(* CoDeSys 2.3 library: oscat270.lib *)
(* Libraries: Standard.lib 22.11.04 11:21:12, SYSLIBCALLBACK.LIB 20.4.05 10:04:48 *)

(* Global variable list: Constants *)
VAR_GLOBAL CONSTANT
	(* setup Parameters *)
	STEP7 : BOOL := FALSE;

	(* Mathematische Konstanten *)
	PI1 : REAL := 3.14159265358979323846264338327950288;	(* Kreiszahl PI *)
	PI2 : REAL := 6.283185307179586476;					(* PI * 2 *)
	E : REAL := 2.71828182845904523536028747135266249;	(* Eulersche Konstante *)

	(* Physikalische Konstanten *)
	C0 : REAL := 299792458 ;							(* Lichtgeschwindigkeit in m/s *)
	EL : REAL := 1.60217653E-19;						(* elementarladung in Colomb = A * s *)
	GN : REAL := 9.80665; 								(* Erdbeschleunigung in m / s² *)
	TK : REAL := -273.15;									(* absoluter Nullpunkt in °C *)
	RU : REAL := 8.314472; 								(*Universelle Gaskonstante in J / (mol · K) *)
	PN : REAL := 101325;									(* NormalDruck in Pa *)

END_VAR

VAR_GLOBAL
END_VAR

(* revisionhistory
hm 3.3.2007
	extended accuracy of pi2
	renamed T0 to Tk for better compatibility with other libraries
	renamed C t0 c0 for better compatibility

hm	2.5.2007
	added RU universal gas constant

hm	1. oct 2007
	added setup parameter STEP7

hm 31. oct 2007
	added PN
*)

(* Data type *)
TYPE esr_data :
STRUCT
	typ : BYTE;
	adress : STRING(10);
	DS : DT;
	TS : TIME;
	data : ARRAY[0..7] OF BYTE;
END_STRUCT
END_TYPE

(* Data type *)
TYPE vector_3 :
STRUCT
	X : REAL;
	Y : REAL;
	Z : REAL;
END_STRUCT
END_TYPE

(* POU _array_init, ST *)
FUNCTION _array_init : BOOL
VAR_INPUT
	pt : POINTER TO ARRAY[0..32000] OF REAL;
	size : INT;
	init : REAL;
END_VAR
VAR
	i: INT;
	stop: INT;
END_VAR


(*
version 1.2	14 nov 2007
programmer 	hugo
tested by		tobias

this function will initialize a given array with a value init.
the function needs to be called:	_array_init(adr("array"),sizeof("array"));
this function will manipulate a given array.
the function manipulates the original array, it rerturnes true when finished.
because this function works with pointers its very time efficient and it needs no extra memory.

*)
stop := SHR(size,2)-1;
FOR i := 0 TO stop DO
	pt^[i] := init;
END_FOR;

_array_init := TRUE;

(* revision History

hm 6.1.2007		rev 1.1
	change type of function to bool
	added  array_init := true to set output true.

hm	14.11.2007	rev 1.2
	changed stop calculation to be more efficient
*)
END_FUNCTION

(* POU _array_median, ST *)
FUNCTION _array_median : REAL
VAR_INPUT
	pt : POINTER TO ARRAY[0..32000] OF REAL;
	size : INT;
END_VAR
VAR
	i: INT;
	stop: INT;
END_VAR

(*
version 1.4	14 nov 2007
programmer 	hugo
tested by		tobias

this function will calculate the median of a given array.
in order to do so the ariginal array is sorted and stays sorted after the function finishes
the function needs to be called:	_array_median(adr("array"),sizeof("array"));
this function will manipulate a given array.
the function will return the median of the original array.
for example [12,0,4,7,1] the median is 4 and the array after the function is called is [0,1,4,7,12]
because this function works with pointers its very time efficient and it needs no extra memory.

*)
_array_sort(pt,size);
stop := SHR(size,2)-1;
IF even(stop) THEN
	_array_median := pt^[stop/2];
ELSE
	i := SHR(stop,1);
	_array_median := (pt^[i] + pt^[i+1]) / 2;
END_IF;

(* old code
stop := (size - SIZEOF(pt)) / SIZEOF(pt);
FOR i := 0 TO stop - 1 DO
	FOR m := i + 1 TO stop DO
		IF pt^[i] > pt^[m] THEN
			temp := pt^[i];
			pt^[i] := pt^[m];
			pt^[m] := temp;
		END_IF;
	END_FOR;
END_FOR;
IF even(stop) THEN
	_array_median := pt^[stop/2];
ELSE
	i := stop/2;
	_array_median := (pt^[i] + pt^[i+1])/2;
END_IF;
*)
(* revision history
hm 	3.3.2007		rev 1.1
	corrected an error, changed the statement line 14	i := TRUNC(stop/2); to i := stop/2;

hm		22. sep 2007	rev 1.2
	changed algorithm to use _array_soft for performance reasons

hm		8. oct 2007		rev 1.3
	deleted unused variables m and temp

hm		14. nov 2007		rev 1.4
	corrected a problem with size calculation
*)
END_FUNCTION

(* POU _array_sort, ST *)
FUNCTION _array_sort : BOOL
VAR_INPUT
	f : POINTER TO ARRAY[1..32000] OF REAL;
	size : INT;
END_VAR
VAR
	i: INT;
	j: INT;
	temp : REAL;
	stop : INT;
	heapsize: INT;
	popmax : REAL;
	size2: INT;
	hs2: INT;
END_VAR

(*
version 1.5	5 jan 2008
programmer 	hugo
tested by		tobias

this function will sort a given array.
the function needs to be called:	_array_sort(adr("array"),sizeof("array"));
this function will manipulate a given array.
the function will not return anything except true, it will instead manipulate the original array.
because this function works with pointers its very time efficient and it needs no extra memory.

*)
(* generate heap *)

size := SHR(size,2);
size2 := SHR(size,1);
FOR i := SIZE2  TO 1 BY -1 DO 		(* zweite Hälfte des Feldes braucht nicht betrachtet werden *)
	j:=i;
    WHILE j <= SIZE2 DO
     	stop := j * 2 + 1;               (* finde Maximum der (beiden) Söhne *)
        IF stop > SIZE THEN stop := stop - 1;
        ELSIF f^[stop-1] > f^[stop] THEN stop := stop - 1;
		END_IF;
        IF f^[j] < f^[stop] THEN   		(* ggf. tauschen *)
         	temp := f^[j];
            f^[j] := f^[stop];
            f^[stop] := temp;
        END_IF;
        j := stop;
    END_WHILE;
END_FOR;

(* heapsort *)
FOR heapsize := size TO 1 BY -1 DO
	popmax := f^[1];
	f^[1] := f^[heapsize];
   	i := 1;
	hs2 := SHR(heapsize,1);
	WHILE i <= hs2 DO	     (* letztes Element an Anfang setzen und versickern lassen *)
       	stop := i * 2 + 1;                (* finde Maximum der (beiden) Söhne *)
        	IF stop > heapsize THEN stop := stop - 1;
        	ELSIF f^[stop-1] > f^[stop] THEN stop := stop - 1;
	 	END_IF;
        	IF f^[i] < f^[stop] THEN	     (* ggf. tauschen *)
            		temp := f^[i];
            		f^[i] := f^[stop];
            		f^[stop] := temp;
        	END_IF;
        	i := stop;
    	END_WHILE;
	f^[heapsize] := popmax;
END_FOR;

_array_sort := TRUE;

(* old algorithm bubble sort used before rev 1.2
stop := (size - SIZEOF(pt)) / SIZEOF(pt);
FOR i := 0 TO stop - 1 DO
	FOR m := i + 1 TO stop DO
		IF pt^[i] > pt^[m] THEN
			temp := pt^[i];
			pt^[i] := pt^[m];
			pt^[m] := temp;
		END_IF;
	END_FOR;
END_FOR;
_array_sort := TRUE;

*)
(* revision history

hm 	6.1.2007 	rev 1.1
	changed return value to true

hm	22. sep 2007	rev 1.2
	changed sorting algorithm to heap sort for performance reasons

hm 	14. nov 2007	rev 1.3
	changed calculation of stop to be more efficient

hm	15 dec 2007		rev 1.4
	added function return true

hm	5. jan 2008		rev 1.5
	improved performance
*)
END_FUNCTION

(* POU even, ST *)
FUNCTION even : BOOL
VAR_INPUT
	in : INT;
END_VAR
VAR
END_VAR


(*
version 1.1	1 dec 2007
programmer 	hugo
tested by		tobias

this function chacks an input for even  value
the output is true if the input is even.
execution time on wago 750 - 841 =  10  us
*)
even := NOT in.0;

(* revision history
hm	1. oct 2006	rev 1.0
	ORIGINAL VERSION
hm	01.12.2007	rev 1.1
	changed code for improoved performance

*)
END_FUNCTION

(* POU acosH, ST *)
FUNCTION acosH : REAL
VAR_INPUT
	X : REAL;
END_VAR
VAR
END_VAR


(*
version 1.1	2 dec 2007
programmer 	hugo
tested by		tobias

this function calculates the arcus cos hyperbolicus

*)
acosH := LN(X + SQRT(X * X - 1));


(* revision history
hm		12 jan 2007	rev 1.0
	original version

hm		2. dec 2007	rev 1.1
	changed code for better performance

*)
END_FUNCTION

(* POU acotH, ST *)
FUNCTION acotH : REAL
VAR_INPUT
	X : REAL;
END_VAR
VAR
END_VAR


(*
version 1.1	5. jan 2008
programmer 	hugo
tested by		tobias

this function calculates the arcus cotangens hyperbolicus

*)
acotH := LN((x+1)/(x-1))*0.5;

(* revision history
hm		12 jan 2007	rev 1.0
	original version

hm		5. jan 2008	rev 1.1
	improved code for better performance
*)
END_FUNCTION

(* POU actuator_2P, ST *)
FUNCTION_BLOCK actuator_2P
VAR_INPUT
	val : REAL;
	force : BOOL;
	force_in : BOOL;
END_VAR
VAR_INPUT CONSTANT
	self_act_time : TIME := t#10d;
	self_act_cycles : INT := 5;
	cycle_time : TIME := t#10m;
	min_ontime : TIME := t#10s;
	min_offtime : TIME := t#10s;
END_VAR
VAR_OUTPUT
	out :BOOL;
	pos : REAL;
END_VAR
VAR
	last_activation : TIME;
	count : INT;
	TON : TIME;
	tx : TIME;
	tc : TIME;
END_VAR


(*
version 1.5	27 dec 2007
programmer 	hugo
tested by		tobias

this is an intelligent actuator interface for any 2point actuator like coil drive.
the 2Point actuator can only switch on/off and therefore a input must be converted to on/off cycles.
the interface can be programmed with double click on the symbol for duty cyle, min_ontime and min_offtime to avoid flickering of the valve or flap.
in addition a self_act_time and self_act_cycles ca be programmed to switch n times on/off every self_act_time to avoid a valve to freeze.
a on and off input can be used to force the valve on or off at all times.
a additional pos output will always indicate the current position of a valve.
the input value must be between 0 and 1.

val		force	force_in	pos	out			
X		0		-			X		duty cycle X
-		1		1			1		1
-		1		0			0		0

*)
(* read system Time *)
tx := DWORD_TO_TIME(T_PLC_MS());
tc := tx - last_activation;

(* verify input to be between 0 and 1 *)
val := LIMIT(0,val,1);

(* check for min ontime or min offtime and wait if not passed *)
IF (out AND tc < min_ontime) OR (NOT out AND tc < min_offtime) THEN RETURN;

(* when force off then shutoff valve *)
ELSIF force AND NOT force_in THEN
	pos := 0;
	out := 0;
	last_activation := tx;
	count := 0;

(* if force on then turn on valve *)

ELSIF force AND force_in THEN
	pos := 1;
	out := 1;
	last_activation := tx;
	count := 0;

(* if nothing happened for self_act_time then do self activation cycles *)
ELSIF (tc >= self_act_time AND count = 0 AND self_act_cycles > 0) OR (count > 0 AND count < self_act_cycles * 2) THEN
	out := NOT out;
	last_activation := tx;
	count := count + 1;
	RETURN;
ELSIF count > 0 THEN
	count := 0;
ELSE
	ton := multime(cycle_time,val);
	IF ton < min_ontime / 2 THEN ton := t#0s; ELSIF ton < min_ontime THEN ton := min_ontime; END_IF;
	IF ton > cycle_time - min_offtime / 2 THEN ton := cycle_time; ELSIF ton > cycle_time - min_offtime THEN ton := cycle_time - min_offtime; END_IF;
	IF ton = t#0s THEN
		IF out =0 THEN
			pos := 0;
			RETURN;
		ELSE
			out := 0;
			pos := 0;
			last_activation := tx;
		END_IF;
	ELSIF ton = cycle_time THEN
		IF out = 1 THEN
			pos := 1;
			RETURN;
		ELSE
			out := 1;
			pos := 1;
			last_activation := tx;
		END_IF;
	END_IF;
	pos := TIME_TO_REAL(ton) / TIME_TO_REAL(cycle_time);
	(* output pulse generation *)
	IF out AND tc >= ton THEN
		out := 0;
		last_activation := tx;
	ELSIF NOT out AND tc >= cycle_time - ton THEN
		out := 1;
		last_activation := tx;
	END_IF;
END_IF;


(*
revision history:

hm		7.10.2006 		rev 1.1
	changed error pos could not reach 1 or 0 under certain conditions due to error in code.
	changed on and off in force and force_in for better usability.

hm		17.1.2007		rev 1.2
	deleted unused variable time_overflow

hm		15.9.2007		rev 1.3
	replaced time() with T_PLC_MS for compatibility and performance reasons

hm		19. 11 2007		rev 1.4
	replaced left over statement time() with tx

hm		27. 12. 2007	REV 1.5
	CHANGED CODE FOR BETTER PERFORMANCE
*)
END_FUNCTION_BLOCK

(* POU cycle_time, ST *)
FUNCTION_BLOCK cycle_time
VAR_INPUT
	rst : BOOL;
END_VAR
VAR_OUTPUT
	ct_min : TIME := t#0s;
	ct_max : TIME := t#0s;
	ct_last : TIME;
	systime : TIME;
	sysdays : INT;
	cycles : DWORD;
END_VAR
VAR
	last_cycle : TIME;
	tx: TIME;
	init: BOOL;
END_VAR


(*
	version 1.2	16 sep 2007
	programmer 	hugo
	tested BY		hans

this function block measures the cycle time and displays the last, min and max cycle time of the current task.
the resolution is 1ms.
the cycles output is a dword counter which counts the cycles.
a rst pulse on the input will reset all data.


*)
tx := DWORD_TO_TIME(T_PLC_MS()) - last_cycle;
IF rst THEN
	ct_min := t#10h;
	ct_max := t#0ms;
	cycles := 0;
ELSIF last_cycle > t#0s THEN
	IF tx < ct_min THEN ct_min := tx;
	ELSIF tx > ct_max THEN ct_max := tx;
	END_IF;
	ct_last := tx;
ELSIF ct_min = t#0s THEN
	ct_min := t#0s - t#1ms;
END_IF;
IF init THEN
	systime := systime + tx;
		IF systime >= t#1d THEN
			systime := systime - t#1d;
			sysdays := sysdays + 1;
		END_IF;
END_IF;
init := TRUE;
last_cycle := last_cycle + tx;
cycles := cycles + 1;

(*	revision history
hm 12.12.2006		rev 1.1
	added cycles output, a dword cycle counter.
hm 10.3.2007			rev 1.2
	changed initialization of ct_min to t#10h for compatibility with siemens s7

hm	16.9.2007		rev 1.2
	changed Time() in T_PLC_MS() for compatibility resons

*)
END_FUNCTION_BLOCK

(* POU T_PLC_MS, ST *)
FUNCTION T_PLC_MS : DWORD
VAR CONSTANT
	debug : BOOL := FALSE;
	N : INT := 0;
	offset : DWORD := 0;
END_VAR
VAR
	tx : TIME;
	temp : DWORD := 1;
END_VAR

(*
version 1.1	12 nov 2007
programmer 	hugo
tested by		tobias

T_PLC_MS reads the internal PLC timer and return the time, it has the advantage to be able to set a debug mode 
and speed up the counter to test the plc timer overrun which occurs every 50 days respectively 25 days at siemens S7
this routine also allows to correct the behavior of s7 where the internal plc counter will not count all 32 bits.

*)
tx := TIME();
T_PLC_MS := TIME_TO_DWORD(Tx);
(* hier muss die korrektur für step7 stattfinden
plctime muss den vollen wertebereich von time ausnutzen:
wenn bei step7 time -24tage bis plus 24 tage ist dann muss der timer auch beim überlauf auf -24tage springen 
und auf keinen fall auf 0 !!!!
für siemens muss ein weiterer fb im main eingebunden werden der sicherstellt das alle 32 bits durchgezählt werden.
es kann nur ein fb sein den er muss sich das oberste (32te) bit merken.
oder etwa spring s7 bei überlauf auf -24 tage????? dann wäre keine korrektur nötig.
*)
IF debug THEN
	T_PLC_MS := (SHL(T_PLC_MS,N) OR SHL(temp,N)-1) + Offset;
END_IF;

(* revision history
hm	14.9.2007	rev 1.0
	original version

hm	12. nov 2007	rev 1.1
	added temporaray variable tx because some compilers could not handle time() as an argument

*)
END_FUNCTION

(* POU Offset, ST *)
FUNCTION Offset : REAL
VAR_INPUT
	X : REAL;
	O1, O2, O3, O4 : BOOL;
	D : BOOL;
END_VAR
VAR_INPUT CONSTANT
	Offset_1 : REAL;
	Offset_2 : REAL;
	Offset_3 : REAL;
	Offset_4 : REAL;
	default : REAL;
END_VAR

(*
version 1.0	12 jan 2007
programmer 	oscat
tested by		tobias

The Function offset adds offsets to an analog signal depending on digital inputs.
all selected offsets are added at the same time.
with the input D a default value instead of the input X can be used.

*) 
IF D THEN Offset := default; ELSE Offset := X; END_IF;
IF O1 THEN Offset := Offset + offset_1; END_IF;
IF O2 THEN Offset := Offset + offset_2; END_IF;
IF O3 THEN Offset := Offset + offset_3; END_IF;
IF O4 THEN Offset := Offset + offset_4; END_IF;
END_FUNCTION

(* POU multime, ST *)
FUNCTION multime : TIME
VAR_INPUT
	t : TIME;
	M : REAL;
END_VAR
VAR
END_VAR


(*
version 1.0	2 oct 2006
programmer 	hugo
tested by		tobias

multiplies a time by a real number and returns a time
*)
multime := REAL_TO_TIME(TIME_TO_REAL(t)*M);
END_FUNCTION

(* POU actuator_3P, ST *)
FUNCTION_BLOCK actuator_3P
VAR_INPUT
	in : REAL;
	force : BOOL;
	on : BOOL;
	end_pos : BOOL;
	diag : BOOL;
END_VAR
VAR_INPUT CONSTANT
	min_ontime : TIME := t#10s;
	min_offtime : TIME := t#10s;
	max_runtime : TIME := t#60s;
	auto_diag_time : TIME := t#10d;
	cal_runtime : TIME := t#600s;
	switch_available: BOOL;
END_VAR
VAR_OUTPUT
	out1 : BOOL;
	out2 : BOOL;
	pos : REAL;
	busy : BOOL;
	error : BOOL;
END_VAR
VAR
	val: REAL;
	tx : TIME;
	last_diag: TIME;
	last : TIME;
	runtime_1 : TIME;
	runtime_2 : TIME;
	state : INT;
	rout: FT_rmp;
	end : R_TRIG;
	cal_timer: TIME;
	Tn: TIME;
END_VAR


(*
version 1.3	 15 sep 2007
programmer 	hugo
tested by		tobias

actuator_3P is an interface for a 3 point actuator.
a 3P actuator is a motor with 2 directions that drives a valve or flap. the position of the valve or flap is controlled by runtime of the motor foreward or backward.
the available inputs are:
in is a real value which specifies the position of the actuator, 0 = 0% and 1 = 100% any value <0 or > 1 is limited to 0 or 1.
a force input must be low for normal operation and if switched high, the motor can only be controlled for 0% or 100% positions with the on input.
an and pos input is available for a end_pos switch, this switch indicates the valve or flap to be at either 0% or 100%
a diag input can at any time start a diag cycle which turns the motor towards the 0% position, then measures the runtime to 100% and then the runtime to 0%
these runtimes are stored and used for absolute positioning of the motor during normal operation.
a setup constand "auto_diag_time can be used to specify how often the actuator repeates this auto_diag cycla automatically.
at power on a cycle is perfomed automatically.
a 0 for this value means auto diag is never performed.

the outputs ar out1 and out2 for up and down direction of the motor. to avoid flickering the output can be programmed for min_ontime and min_offtime.
a pos outout indicates the absulute position of the actuator during operation and a busy output indicates the actuator is busy.
a error output is initiated when the specified max_runtime is reached by any direction during debug.
also when the up and down direction differs by more then 10% the error output is set.

for absolute positioning accuracy the actuator has a setup variable "cal_runtime" if this is set the actuator measures the total runtime of the motors and when this 
cal_runtime is exceeded it resets the actuator to 0% position and sets the output again to assure absolute accuracy.

autodiag and calibration can be shut off by setting the appropriate values to 0.
a switch_available setup variable specifies if end_pos switches are available.

*)
(* setup *)
Tn := DWORD_TO_TIME(T_PLC_MS());
tx := Tn - last;
end(clk := end_pos);

(* init only when first started *)
IF state = 0 THEN
	runtime_1 := max_runtime;
	runtime_2 := max_runtime;
	state := 1;
	rout(KR := 1000 / TIME_TO_REAL(runtime_1), KF := 1000 / TIME_TO_REAL(runtime_1) );
	tx := t#0s;
	last := Tn;
	last_diag := last;
END_IF;

(* check for end_sw and stop if reached *)
IF switch_available AND out1 AND end.Q THEN
	(* upper limit has been reached *)
	out1 := 0;
	rout(rmp := 0, in := 1);
	rout.Rmp := 1;
ELSIF switch_available AND out2 AND end.Q THEN
	(* lower limit has been reached *)
	out2 := 0;
	rout(rmp := 0, in := 0);
	rout.Rmp := 1;
END_IF;

(* check for min_offtime and min_ontime and return if it has not elapsed *)
IF NOT busy AND tx < min_offtime THEN RETURN;
ELSIF busy AND tx < min_ontime THEN RETURN;

(* check for last diag cycle and start diag if auto_diag_time has elapsed *)
ELSIF (tn - last_diag > auto_diag_time AND state > 10 AND auto_diag_time > t#0s) OR (diag AND state >= 10) THEN state := 1;

(* check if force pin is high *)
ELSIF force THEN state := 10;

(* check if calibration is necessary *)
ELSIF cal_timer > cal_runtime AND state = 99 AND cal_runtime > t#0s THEN state := 20;
END_IF;

(* state machine for operation *)
CASE state OF

1 :	(* diagnostic start *)
	(* all data is reset and out2 is turned on to make sure we start from top position *)
	last_diag := tn;
	diag := 0;
	state := 2;
	pos := 0;
	busy := 1;
	last := tn;
	out1 := 0;
	out2 := 1;
	RETURN;

2:	(* wait for max_runtime or end_pos to be reached *)
	IF tx < max_runtime AND NOT end.Q THEN RETURN; END_IF;
	state := 3;
	last := tn;
	out1 := 1;
	out2 := 0;
	RETURN;

3: 	(* measure runtime_2 *)
	IF tx < max_runtime AND NOT end.Q THEN RETURN; END_IF;
	state := 4;
	runtime_1 := tx;
	last := tn;
	out1 := 0;
	out2 := 1;
	RETURN;

4:	(* measure runtime_1 *)
	IF tx < max_runtime AND NOT end.Q THEN RETURN; END_IF;
	state := 99;
	runtime_2 := tx;
	last := tn;
	out2 := 0;
	busy := 0;
	(* reset the output ramp generator to the 0% position as the valve is after diags *)
	rout(rmp := 0, in := 0);
	rout.Rmp := 1;
	cal_timer := t#0s;
	IF differ(TIME_TO_REAL(runtime_1), TIME_TO_REAL(runtime_2), TIME_TO_REAL(max_runtime) * 0.1) THEN error := TRUE;
	ELSIF runtime_1 > multime(max_runtime, 0.9) AND switch_available THEN error := TRUE;
	ELSIF runtime_2 > multime(max_runtime, 0.9) AND switch_available THEN error := TRUE;
	END_IF;
	RETURN;

10: (* force pin is active, outputs are forced on or off by the on pin *)
	IF on AND NOT out2 THEN val := 1;
	ELSIF NOT on AND NOT out1 THEN val := 0;
	END_IF;
	IF NOT force THEN state := 99; END_IF;

20 : (* calibrate to allow for correction of positioning error addig up *)
	cal_timer := t#0s;
	state := 21;
	pos := 0;
	busy := 1;
	last := tn;
	out1 := 0;
	out2 := 1;
	RETURN;

21:	(* after end_sw or max_runtime we can be sure to have reached the 0% position *)
	IF tx < max_runtime AND NOT end.Q THEN RETURN; END_IF;
	state := 99;
	out2 := 0;
	busy := 0;
	last := tn;
	rout(rmp := 0, in := 0);
	rout.Rmp := 1;
	RETURN;

99: (* normal operation *)
	(* only if input changes for an equivalent of min_ontime then change the output *)
	(* if there is a directional change then wait until last step is finished *)
	IF in < TIME_TO_REAL(min_ontime)/TIME_TO_REAL(max_runtime)/2 THEN val := 0;
	ELSIF in > 1 - TIME_TO_REAL(min_ontime)/TIME_TO_REAL(max_runtime)/2 THEN val := 1;
	ELSIF differ(LIMIT(0,in,1), val, TIME_TO_REAL(min_ontime) / TIME_TO_REAL(max_runtime)) OR in = 0 OR in = 1 THEN
		IF in < val AND NOT out1 THEN val := in;
		ELSIF in > val AND NOT out2 THEN val := in;
		END_IF;
	END_IF;

END_CASE;

(* output ramp generator *)
rout(in := val);
out1 := rout.busy AND rout.UD;
out2 := rout.busy AND NOT rout.UD;
pos := rout.out;

(* set the busy output and if busy goes low, then set the last time in order to check for min_offtime *)
IF NOT busy AND rout.busy THEN
	last := tn;
ELSIF busy AND NOT rout.busy THEN
	cal_timer := cal_timer + tx;
	last := tn;
END_IF;
busy := rout.busy;



(* revision history

19.10.2006	rev 1.1
	added security checks for end_switch to avoid overrun of the end_switch, hans

23.1.2007		rev 1.2
	deleted unused variables force_on and force_off

15.9.2007	hm	rev 1.3
	replaced Time() with T_PLC_MS for compatibility and performance reasons

*)
END_FUNCTION_BLOCK

(* POU FT_rmp, ST *)
FUNCTION_BLOCK FT_rmp
VAR_INPUT
	Rmp : BOOL := TRUE;
	in : REAL;
	KR : REAL;
	KF : REAL;
END_VAR
VAR_OUTPUT
	out : REAL;
	busy : BOOL;
	UD : BOOL;
END_VAR
VAR
	tx: TIME;
	last: TIME;
	init: BOOL;
END_VAR

(*
	version 1.4	25 jan 2008
	programmer 	oscat
	tested BY		oscat

this ramp function follows an input signal with a linear ramp up or down, the up or down speed can be set with KF and KR.
a K factor of 1 means 1 unit per second on the output. K factors can only be positive and not negative.
a busy output signals the ramp is running or busy false means the in value is present on the output.
a rmp input false means the output follows the input dierctly while a rmp = true means the output follows the input with a ramp.
a updn output signal the directon of the ramp (up or down).

*)
(* read system time *)
tx := DWORD_TO_TIME(T_PLC_MS()) - last;

IF NOT init THEN
	init := TRUE;
	last := tx;
	tx := t#0s;
	out := in;
END_IF;
IF NOT rmp THEN
	out := in;
	busy := FALSE;
ELSIF out > in THEN
	(* ramp down *)
	out := out - TIME_TO_REAL(tx) * 0.001 * KF;
	out := MAX(in, out);
ELSIF out < in THEN
	(* ramp up *)
	out := out + TIME_TO_REAL(tx) * 0.001 * KR;
	out := MIN(in, out);
END_IF;

(* set busy and dir flags *)
IF out < in THEN
	busy := TRUE;
	ud := 1;
ELSIF out > in THEN
	busy := TRUE;
	ud := 0;
ELSE
	busy := FALSE;
END_IF;
last := last + tx;


(* revision history:

hm 8.10.2006			rev 1.1
	added ud output

hm 12. feb 2007		rev 1.2
	added init variable and corrected a possible startup problem

hm	17. sep 2007	rev 1.3
	replaced time() with t_plc_ms() for compatibility reasons

hm	25. jan 2008	rev 1.4
	performance improvements
	allow KR and KF to be 0
*)
END_FUNCTION_BLOCK

(* POU differ, ST *)
FUNCTION differ : BOOL
VAR_INPUT
	in1 : REAL;
	in2 : REAL;
	X : REAL;
END_VAR
VAR
END_VAR

(*
version 1.0	8 oct 2006
programmer 	hugo
tested by		tobias

this function checks if in1 differs more then x from in2
the output is true if in1 < in2 - x or in1 > in2 + X
*)
differ := in1 < in2 - X OR in1 > in2 + X;
END_FUNCTION

(* POU actuator_pump, ST *)
FUNCTION_BLOCK actuator_pump
VAR_INPUT
	in : BOOL;
	manual : BOOL;
	rst : BOOL := FALSE;
END_VAR
VAR_INPUT CONSTANT
	min_ontime : TIME := t#10s;
	min_offtime : TIME := t#10s;
	run_every : TIME := t#10000m;
END_VAR
VAR_OUTPUT
	pump : BOOL;
	runtime : REAL;
	cycles : REAL;
END_VAR
VAR
	tx : TIME;
	last_change : TIME;
	meter : ontime;
	old_man : BOOL;
	init: BOOL;
END_VAR

(*
	version 1.2	15 sep 2007
	programmer 	oscat
	tested BY		oscat

actuator_pump is a pump interface which can be controlled by an input in and an input manual.
in or manual high turns the pump output on.
a rst input is used to reset the runtime counters.
when the pump was not active for a time run_every the actuator turns on the pump automatically for min_ontime.
two setup variables min_ontime and min_offtime guarantee a minimum runtime and offtime of the pump.
the units are hours and the output type is real to prevent from overfow.

*)
tx := DWORD_TO_TIME(T_PLC_MS());

IF NOT init THEN
	init := TRUE;
	last_change := tx;
ELSIF rst THEN
	rst := FALSE;
	meter(rst := TRUE);
	meter.rst := FALSE;
ELSIF manual AND NOT pump AND NOT old_man THEN
	last_change := tx;
	pump := TRUE;
ELSIF NOT manual AND old_man AND pump AND NOT in THEN
	last_change := tx;
	pump := FALSE;
ELSIF in AND NOT pump AND tx - last_change >= min_offtime THEN
	last_change := tx;
	pump := TRUE;
ELSIF pump AND NOT in AND NOT manual AND tx - last_change >= min_ontime THEN
	last_change := tx;
	pump := FALSE;
ELSIF NOT pump AND tx - last_change >= run_every THEN
	last_change := tx;
	pump := TRUE;
END_IF;

meter(in := pump);
runtime := meter.ontime;
cycles := meter.cycles;
old_man := manual;

(*
27.12.2006	rev 1.1	hm
	fixed a failure while the pump would run for tmin after startup.

15.9.2007	hm	rev 1.2
	replaced Time() with T_PLC_MS for compatibility and performance reasons

*)
END_FUNCTION_BLOCK

(* POU Meter, ST *)
FUNCTION_BLOCK Meter
VAR_INPUT
	M1, M2 : REAL;
	I1, I2 : BOOL;
	D : REAL := 1;
	RST : BOOL;
END_VAR
VAR_OUTPUT RETAIN
	MX : REAL;
END_VAR
VAR
	int1 : FT_INT;
	int2 : FT_INT;
END_VAR

(*
	version 1.1	8. feb 2008
	programmer 	oscat
	tested BY		oscat

METER measures usage of power or similar values the output MX is the summ of the inputs over time.
MX := sum over time of I1 * P1 + I2 * P2.
a simple example is the consumption counter for a 2 stage oil burner where stage 1 is 10KW and stage 2 is 20KW.
I1 and I2 decide which value is accounted for, I1 = True only counts P1, I2 is True counts P2 
and I1 and I2 is true counts P1 and P2.
the meter can be used for all kind of consumption meters. P1 and P2 can change on the fly.

*)
(* meter would have a problem when int1 or int2 reach big values
and a short time tick would add a value smaller then the 7 digit resolution of real
therefore the variables m1 and m2 are used to store the counted values 
while the integrators are kept at small values to avoid this overrun
*)

int1(in := M1, Run := I1, rst := rst);
int2(in := M2, Run := I2, rst := rst);
MX := (int1.Out+ int2.Out) / D;

(* revision history

hm	16. sep.2007		rev 1.0
	original version

hm	7. feb 2008		rev 1.1
	use new version of ft_int to avoid a counting stop at high values
	deleted unnecessary limits
*)
END_FUNCTION_BLOCK

(* POU FT_INT, ST *)
FUNCTION_BLOCK FT_INT
VAR_INPUT
	in : REAL;
	K : REAL := 1;
	run : BOOL := 1;
	rst: BOOL := 0;
	out_min : REAL := -1E-37;
	out_max : REAL := 1E37;
END_VAR
VAR_OUTPUT
	Out : REAL;
END_VAR
VAR
	last: DWORD;
	in_last : REAL;
	tx: DWORD;
	init: BOOL;
	tc: DWORD;
	out1: REAL;
	out2: REAL;
	tmp: REAL;
END_VAR


(*
version 1.7	8. feb 2008
programmer 	hugo
tested by		tobias

FT_int is an integrator with input IN and factor K.
integration is only done while run = true, if run is false integration is stopped and the out remains at the last value.
if run is left unconnected, run is considered true by the function block.
the output ET will display the total integration time from last reset.
a rst input will reset output and the timer ET to 0.
the out_min and out_max values can be set to ,imit the output value range. 
the default for K is 1.

 
*)
(* read and store system time *)
tx := T_PLC_US();
tc := tx - last;

(* startup initialisation *)
IF rst OR NOT init THEN
	out1 := 0;
	out2 := 0;
	init := TRUE;
	last := tx;
ELSIF run AND tc > 0 THEN
	last := tx;
	out1 := out1 + (in + in_last) * tc * K * 5E-7;
	tmp := in * K * 10000;
	IF out1 > tmp THEN
		out1 := out1 - tmp;
		out2 := out2 + tmp;
	END_IF;
ELSIF NOT run THEN
	last := tx;
END_IF;
in_last := in;
out := LIMIT(out_min, out1 + out2, out_max);

(*
hm 13.12.2006	rev 1.1
	changed to "trapezregel" which increases accuracy
	before out := out + in * time new: out := out + (in + in_last) / 2 * time

hm 15.1.2007		rev 1.2
	added default for k to be 1.

hm	15.9.2007		rev 1.3
	replaced time() with T_PLC_US for compatibility and performance reason
	increased internal accuracy to microseconds

hm 29. oct 2007		rev 1.4
	changed code so int will not be called is time difference is 0 to increase accuracy on systems
	with cycle times below 1ms

hm	2. dec 2007	 	rev 1.5
	changed code for better performance

hm	5. jan 2008		rev 1.6
	further improvements in performance

hm	8. feb 2008		rev 1.7
	deleted limits +/- 1000 now limit is the range of real
	added variables out1 and out2 to extend the resolution
	corrected an error with elapsed time
	deleted unusfull output ET
*)
END_FUNCTION_BLOCK

(* POU T_PLC_US, ST *)
FUNCTION T_PLC_US : DWORD
VAR CONSTANT
	debug : BOOL := FALSE;
	N : INT := 0;
	offset : DWORD := 0;
END_VAR
VAR
	tx : TIME;
	temp : DWORD := 1;
END_VAR

(*
version 1.1	12 nov 2007
programmer 	hugo
tested by		tobias

T_PLC_US reads the internal PLC timer and return the time, it has the advantage to be able to set a debug mode 
and speed up the counter to test the plc timer overrun which occurs every 50 days respectively 25 days at siemens S7
this routine also allows to correct the behavior of s7 where the internal plc counter will not count all 32 bits.

*)
tx := TIME();
T_PLC_US := TIME_TO_DWORD(Tx)*1000;
(* hier muss die korrektur für step7 stattfinden
plctime muss den vollen wertebereich von time ausnutzen:
wenn bei step7 time -24tage bis plus 24 tage ist dann muss der timer auch beim überlauf auf -24tage springen 
und auf keinen fall auf 0 !!!!
für siemens muss ein weiterer fb im main eingebunden werden der sicherstellt das alle 32 bits durchgezählt werden.
es kann nur ein fb sein den er muss sich das oberste (32te) bit merken.
oder etwa spring s7 bei überlauf auf -24 tage????? dann wäre keine korrektur nötig.
*)
IF debug THEN
	T_PLC_US := (SHL(T_PLC_US,N) OR SHL(temp,N)-1) + Offset;
END_IF;

(* revision history
hm	14.9.2007	rev 1.0
	original version

hm	12. nov 2007	rev 1.1
	added temporaray variable tx because some compilers could not handle time() as an argument

*)
END_FUNCTION

(* POU ontime, ST *)
FUNCTION_BLOCK ontime
VAR_INPUT
	in : BOOL;
	rst : BOOL := FALSE;
END_VAR
VAR_OUTPUT RETAIN
	ontime : REAL;
	last_on : REAL;
	cycles : REAL;
END_VAR
VAR
	tx: DWORD;
	last : DWORD;
	edge : BOOL := 0;
	L_time1, H_time1, L_time2, H_time2 : DWORD;
	temp: DWORD;
END_VAR

(*
version 1.4	2 dec 2007
programmer 	oscat
tested by		tobias

M_runtime measures the ontime of a signal in hours.
the output is of type real because the time type will overflow within 49 days.
the units are hours.

*)
(* read system time *)
tx := T_PLC_MS();

IF rst THEN
	L_time1 := 0;
	H_time1 := 0;
	cycles := 0;
	L_time2 := 0;
	H_time2 := 0;
	ontime := 0;
	last_on := 0;
ELSIF in THEN
	temp := L_time1;
	L_time1 := L_time1 + (tx-last);
	IF temp > L_time1 THEN H_time1 := H_time1 + 1; END_IF;
	ontime := L_time1/3600000.0 + 1193.046471 * H_time1;
	temp := L_time2;
	L_time2 := L_time2 + (tx-last);
	IF temp > L_time2 THEN H_time2 := H_time2 +2; END_IF;
	last_on := L_time2/3600000.0 + 1193.046471 * H_time2;
	IF NOT edge THEN
		cycles := cycles +1;
		last_on := 0;
		L_time2 := 0;
		H_time2 := 0;
	END_IF;
END_IF;
last := tx;
edge := in;

(* revision history
hm 22.2.2007		rev 1.1
	changed VAR RETAIN PERSISTENT to VAR RETAIN for better compatibility
	wago lon contollers do not support persisitent

hm 2.8.2007		rev 1.2
	adding time up in a real number will automatically lead to the point where 
	small time scales like the cycle time will be below the resolution of real and therefore
	ontime would not increase in small steps as necessary
	the time is now measured internally in two  dwords and be converted to real only for
	output purposes.
	deleted the variable power because it was unnecessary

hm	16.9.2007	rev 1.3
	changes time() to T_plc_ms() for compatibility reasons

hm	2. dec. 2007	rev 1.4
	chaged code for better performance
*)
END_FUNCTION_BLOCK

(* POU actuator_UD, ST *)
FUNCTION_BLOCK actuator_UD
VAR_INPUT
	UD : BOOL;
	ON : BOOL;
	Manual : BOOL := 0;
	Up : BOOL;
	Dn : BOOL;
	off : BOOL := 0;
	YUP_in : BOOL;
	YDN_in : BOOL;
END_VAR
VAR_INPUT CONSTANT
	TON : TIME;
	TOFF : TIME;
	out_return : BOOL;
END_VAR
VAR_OUTPUT
	Yup : BOOL;
	Ydn : BOOL;
	status : BYTE;
END_VAR
VAR
	tx : TIME;
	last : TIME;
	init: BOOL;
END_VAR

(*
version 1.2	15 sep 2007
programmer 	hugo
tested by		tobias

out_ud is a up/dn or Right/left locked output driver.
it can be controlled by automatic inputs UD and ON as well as manual inputs for up and dn.
a security input to shut off at any time is prvided by the off input.
two time set inputs ton and toff specify a minimum on time for outputs and a minimum off time before the next output can become active.
the module assures that only one output can be active at any time.
for higher security pls make sure you use hardware locking of the outputs to prevent from defective wiring or outputs.
further security is provided b feedback inputs Yup_in and Ydn_in which are separate inputs for the output signal, if these inputs are not available 
pls connect them directly to Yup and Ydn.
manual mode will override automatic mode by setting the manual input high.
a status output will be 0 for normal operation or 1 - 99 for error reporting and 101 - 199 for status reporting
The status output is ESR comptible.
*)
(* read system time *)
tx := DWORD_TO_TIME(T_PLC_MS());

IF NOT init THEN
	(* INITIALIZATION AT FIRST CALL *)
	last := tx;
	init := TRUE;
ELSIF off THEN
	(* emergency shut off detected *)
	Yup := FALSE;
	Ydn := FALSE;
	last := tx;
	status := 101;

(* WATH FOR MIN TON TIME *)
ELSIF ((Yup OR Ydn) AND tx - last < Ton) THEN RETURN;
ELSIF NOT yup AND NOT ydn AND tx - last < toff THEN	RETURN;

(* manual operation *)
ELSIF manual THEN
	status := 102;
	(* directional chage set both outs 0 first *)
	IF yup AND NOT up OR ydn AND NOT dn THEN
		ydn := FALSE;
		yup := FALSE;
		last := tx;
	(* manual up operation *)
	ELSIF UP AND NOT DN AND NOT OFF THEN
		Ydn := FALSE;
		Yup := TRUE;
		last := tx;
		status := 103;
	(* manual down operation *)
	ELSIF DN AND NOT UP AND NOT OFF THEN
		Yup := FALSE;
		Ydn := TRUE;
		last := tx;
		status := 104;
	(* maual mode but no up or down *)
	ELSE
		IF YUP OR YDN THEN LAST := tx; END_IF;
		Yup := FALSE;
		Ydn := FALSE;
	END_IF;

(* automatic operation *)
ELSE
	(* directional change set outputs low first *)
	IF yup AND NOT ud OR ydn AND UD THEN
		yup := FALSE;
		ydn := FALSE;
		last := tx;
	(* automatic up operation *)
	ELSIF Ud AND on AND NOT OFF THEN
		Ydn := FALSE;
		Yup := TRUE;
		last := tx;
		status := 111;

	(* automatic down operation *)
	ELSIF NOT UD AND on AND NOT OFF THEN
		Yup := FALSE;
		Ydn := TRUE;
		last := tx;
		status := 112;
	(* standby mode *)
	ELSE
		IF Yup OR Ydn THEN last := tx; END_IF;
		Yup := FALSE;
		Ydn := FALSE;
		status := 110;
	END_IF;
END_IF;

(* make sure Yup and Ydn are never on at the same time *)
IF Ydn AND Yup_in AND out_return THEN
	Ydn := FALSE;
	status := 1;
END_IF;
IF Yup AND Ydn_in AND out_return THEN
	Yup := FALSE;
	status := 2;
END_IF;

(* revision history
hm 22. jan 2007	rev 1.1
	added status output
	changed inputs ton, toff to config variables
	added config var out_return to enable yup_in and Ydn_in
	manual mod will override automatic mode 

hm	15.9.2007	rev 1.2
	replaced Time() with T_PLC_MS for compatibility and performance reasons
*)
END_FUNCTION_BLOCK

(* POU AIN, ST *)
FUNCTION AIN : REAL
VAR_INPUT
	in : DWORD;
END_VAR
VAR_INPUT CONSTANT
	Bits : BYTE;
	sign : BYTE := 255;
	low : REAL := 0;
	high : REAL := 10;
END_VAR
VAR CONSTANT
	ff : DWORD := 16#FFFFFFFF;
END_VAR
VAR
	temp1 : DWORD;
	temp2 : DWORD;
	sx : BOOL;
END_VAR

(*
version 1.4	2 dec 2007
programmer 	oscat
tested by		tobias

Ain converts signals from A/D converters or other analog sources to an internal real value
the lowest number of bits are extracted from the input word and the sign will be extracted if available separately.
the output signal is then conditioned to range from low to high values for a 0 to max value on the analog inputs:
for example a 15bit input (bits := 12) with sign at bit 15 (0..15) will deliver 0.0 (low value at 0) for an input value of 2#0000_0000_0000
an input value of 2#1111_1111_1111 will deliver 10.0 on the output (high value set to 10).

*) 
(* extract the sign bit *)
IF sign < 32 THEN
	temp1 := SHR(in,sign);
	sx := temp1.0;
ELSE
	sx := FALSE;
END_IF;
temp1 := SHR(ff,32-bits);
temp2 := in AND temp1;
AIN := (high - low)*temp2 / temp1 + low;
IF sx THEN AIN := -AIN; END_IF;

(* revision history
hm 18.8.2006	rev 1.1
	fixed an error with low value negative and high value 0.

hm 19.1.2007	rev 1.2
	fixed an error with sign bit.

hm	13.9.2007	rev 1.3
	changed code to avoid warning under codesys 2.8.1

hm	2. dec 2007	rev 1.4
	changed code for better performance
*)
END_FUNCTION

(* POU Air_density, ST *)
FUNCTION Air_density : REAL
VAR_INPUT
	T : REAL;
	P : REAL;
	RH : REAL;
END_VAR
VAR CONSTANT
	RL : REAL := 287.05;
	RX : REAL := 3.773319E-3;
END_VAR
VAR
END_VAR

(*
version 1.1	4 dec 2007
programmer 	hugo
tested by		tobias

this function calculates the air density between 0 and 100 deg C

*)
Air_density := PN * (1 - RH * SDD(T, TRUE) * RX / P) / (RL * ( T - TK));

(* original code used for rev 1.0

SDD := SDD(T,FALSE);
RF := RL / (1- RH*SDD/P*RX);
Air_density := P / (RF * (T-TK));

*)

(* revision history

hm	29.10.2007		rev 1.0
	original version

hm	4.12.2007		rev 1.1
	changed code for better performance

*)
END_FUNCTION

(* POU SDD, ST *)
FUNCTION SDD : REAL
VAR_INPUT
	T : REAL;
	ICE: BOOL;
END_VAR
VAR CONSTANT
END_VAR
VAR
END_VAR

(*
version 1.1	2 dec 2007
programmer 	hugo
tested by		tobias

this function calculates the vapor saturation pressure for moist Air over ice or water

*)
IF ice THEN
	SDD := 611.153 * EXP(22.4433 * T / (272.186 + T));
ELSE
	SDD := 611.213 * EXP(17.5043 * T / (241.2 + T));
END_IF;

(* old code used in rev 1.0
IF ice THEN
	SDD := 611.153 * exp10(9.747*T / (272.186 + T));
ELSE
	SDD := 611.213 * exp10(7.602*T / (241.2 + T));
END_IF;
*)


(* revision history

hm 29 oct 2007		rev 1.0
	original version

hm	2. dec 2007		rev 1.1
	changed code for better performance
*)
END_FUNCTION

(* POU Air_enthalpy, ST *)
FUNCTION Air_enthalpy : REAL
VAR_INPUT
	T : REAL;
	RH : REAL;
END_VAR
VAR CONSTANT
	CPL : REAL := 1.00482;
	CW : REAL := 1.86;
	LH : REAL := 2500.78;
END_VAR
VAR
END_VAR

(*
version 1.1	2 nov 2007
programmer 	hugo
tested by		tobias

this function calculates the enthalpy for humid air between 0 and 100 deg C

*)
Air_enthalpy := CPL * T + (CW * T + LH) * dew_con(RH,T);

(* revision history

hm	31.10.2007		rev 1.0
	original version

hm	2.11.2007		rev 1.1
	deleted unused variable RF

hm	2.12.2007		rev 1.2
	changed code for better performance
*)
END_FUNCTION

(* POU dew_con, ST *)
FUNCTION dew_con : REAL
VAR_INPUT
	RH : REAL;
	T : REAL;
END_VAR
VAR CONSTANT
END_VAR
VAR
END_VAR

(*
version 1.2	2 dec 2007
programmer 	hugo
tested by		tobias

this function calculates the water concentratin in air for a given temperature and relative humidity.
the output states the concentration of water vapor in air in Gramms / qubic meter.

*)
IF rh > 0 THEN
(*	this code is good to read but need to be improoved
	SDD := 6.1078*EXPT(10,(a*T)/(b+T));
	DD := RH/100 * SDD;
	V := LOG(DD/6.1078);
	TD := b*V/(a-v);
	dew_con := 0.1 * mw / RU * DD / (T - TK);
*)
	dew_con := 2.166824303E-2 * RH * SDD(T,FALSE)  / (T - TK);
ELSE
	dew_con := 0;
END_IF;

(*
Bezeichnungen:
r = relative Luftfeuchte
T = Temperatur in °C
TK = Temperatur in Kelvin (TK = T + 273.15)
TD = Taupunkttemperatur in °C
DD = Dampfdruck in hPa
SDD = Sättigungsdampfdruck in hPa

Parameter:
a = 7.5, b = 237.3 für T >= 0
a = 7.6, b = 240.7 für T < 0 über Wasser (Taupunkt)
a = 9.5, b = 265.5 für T < 0 über Eis (Frostpunkt)

R* = 8314.3 J/(kmol*K) (universelle Gaskonstante)
mw = 18.016 kg (Molekulargewicht des Wasserdampfes)
AF = absolute Feuchte in g Wasserdampf pro m3 Luft

Formeln:

   1. SDD(T) = 6.1078 * 10^((a*T)/(b+T))
   2. DD(r,T) = r/100 * SDD(T)
   3. r(T,TD) = 100 * SDD(TD) / SDD(T)
   4. TD(r,T) = b*v/(a-v) mit v(r,T) = log10(DD(r,T)/6.1078)
   5. AF(r,TK) = 10^5 * mw/R* * DD(r,T)/TK; AF(TD,TK) = 10^5 * mw/R* * SDD(TD)/TK 

*)

(* revision history

hm 29 apr 2007		rev 1.0
	original version

hm	13.sep 2007		rev 1.1
	improoved coding for speed
	deleted unused variabled SDD,DD,V, TD

hm	2. dec 2007		rev 1.2
	changed code for better performance
	output is now in Gramms / Qubic meter
*)
END_FUNCTION

(* POU Aout, ST *)
FUNCTION Aout : DWORD
VAR_INPUT
	in : REAL;
END_VAR
VAR_INPUT CONSTANT
	Bits : BYTE;
	sign : BYTE := 255;
	low : REAL := 0;
	high : REAL := 10;
END_VAR
VAR CONSTANT
	ff : DWORD := 2#1;
END_VAR
VAR
	in2 : REAL;
	sx : BOOL;
END_VAR

(*
version 1.3	2 dec 2007
programmer 	oscat
tested by		tobias

this module conditions an internal real value for a signal output D/A converter.
Aout converts and internal real value to a word for an D/A converter or other output devices.
The input value is converted to a n-bit wide output and a sign bit is set separately as specified.
the outout min value is set for the specified min input value and the max output is set for the max input value.
an input higher or lower then the max or min value will set the respective max or min value or the output.


*) 
(* if sign bit is defined *)
IF sign < 32 THEN
	sx := sign_R(in);
	in2 := ABS(in);
ELSE
	in2 := in;
END_IF;

(* begrenze in auf die zulässigen werte *)
IF in2 < low THEN
	in2 := low;
ELSIF in2 > high THEN
	in2 := high;
END_IF;

(* Berechne den Ausgnagswert *)
Aout := REAL_TO_DWORD((in2 - low) / (high - low) * (SHL(ff,bits) -1));
IF sx THEN Aout := SHL(ff,sign) OR Aout; END_IF;

(*
revision history

hm 18.1.2007		rev 1.1
	renamed Modul to aout.
	changed Output to 32 Bit max.
	corrected error with sign bit.

hm	13.9.2007	rev 1.2
	changed code to avoid warning under codesys 2.8.1

hm	2. dec 2007	rev 1.3
	changed code for better performance
*)
END_FUNCTION

(* POU sign_R, ST *)
FUNCTION sign_R : BOOL
VAR_INPUT
	in : REAL;
END_VAR
VAR
	ptr : POINTER TO DWORD;
END_VAR

(*
version 1.2	1 dec 2007
programmer 	hugo
tested by	tobias

this function return true if the real input is negative

*)
ptr := ADR(in);
sign_R := ptr^.31;



(* revision history
hm 19.1.2007	rev 1.1
	changed method of function for better compatibility to other systems

hm	1.12.2007	rev 1.2
	changed code to improve performance
*)
END_FUNCTION

(* POU array_avg, ST *)
FUNCTION array_avg : REAL
VAR_INPUT
	pt : POINTER TO ARRAY[0..32000] OF REAL;
	size : INT;
END_VAR
VAR
	i: INT;
	stop: INT;
END_VAR

(*
version 1.1	12 dec 2007
programmer 	hugo
tested by		tobias

this function will calculate the average of a given array.
the function needs to be called:	array_avg(adr("array"),sizeof("array"));
because this function works with pointers its very time efficient and it needs no extra memory.

*)
stop := SHR(size,2)-1;
array_avg := pt^[0];
FOR i := 1 TO stop DO
	array_avg := array_avg + pt^[i];
END_FOR;
array_avg := array_avg / (stop + 1);


(* revision history
hm	2. oct 2007	rev 1.0
	original version

hm	12. dec 2007	rev 1.1
	chaged code for better performance

*)
END_FUNCTION

(* POU array_max, ST *)
FUNCTION array_max : REAL
VAR_INPUT
	pt : POINTER TO ARRAY[0..32000] OF REAL;
	size : INT;
END_VAR
VAR
	i: INT;
	stop: INT;
END_VAR

(*
version 1.0	2 oct 2006
programmer 	hugo
tested by		tobias

this function will calculate the max value of a given array.
the function needs to be called:	array_max(adr("array"),sizeof("array"));
because this function works with pointers its very time efficient and it needs no extra memory.

*)
stop := (size -SIZEOF(pt)) / SIZEOF(pt);
array_max := pt^[0];
FOR i := 1 TO stop DO
	IF pt^[i] > array_max THEN array_max := pt^[i]; END_IF;
END_FOR;
END_FUNCTION

(* POU array_min, ST *)
FUNCTION array_min : REAL
VAR_INPUT
	pt : POINTER TO ARRAY[0..32000] OF REAL;
	size : INT;
END_VAR
VAR
	i: INT;
	stop: INT;
END_VAR

(*
version 1.0	2 oct 2006
programmer 	hugo
tested by		tobias

this function will calculate the min value of a given array.
the function needs to be called:	array_min(adr("array"),sizeof("array"));
because this function works with pointers its very time efficient and it needs no extra memory.

*)
stop := (size - SIZEOF(pt)) / SIZEOF(pt);
array_min := pt^[0];
FOR i := 1 TO stop DO
	IF pt^[i] < array_min THEN array_min := pt^[i]; END_IF;
END_FOR;
END_FUNCTION

(* POU array_sdv, ST *)
FUNCTION array_sdv : REAL
VAR_INPUT
	pt : POINTER TO ARRAY[0..32000] OF REAL;
	size : INT;
END_VAR
VAR
END_VAR

(*
version 1.0	1 apr 2007
programmer 	hugo
tested by		tobias

this function will calculate the standard deviation of a given array.
the function needs to be called:	array_sdv(adr("array"),sizeof("array"));
because this function works with pointers its very time efficient and it needs no extra memory.

*)
(* standard deviation is simply the square root of the variance *)

array_sdv := SQRT(array_var(pt, size));

(* revision history
hm 1.4.2007	rev 1.0
	function created
*)
END_FUNCTION

(* POU array_var, ST *)
FUNCTION array_var : REAL
VAR_INPUT
	pt : POINTER TO ARRAY[0..32000] OF REAL;
	size : INT;
END_VAR
VAR
	avg : REAL;
	i: INT;
	stop: INT;
END_VAR

(*
version 1.1	12 dec 2007
programmer 	hugo
tested by		tobias

this function will calculate the variance of a given array.
the function needs to be called:	array_var(adr("array"),sizeof("array"));
because this function works with pointers its very time efficient and it needs no extra memory.

*)
(* at first we calualte the arithmetic average of the array *)

stop := SHR(size,2)-1;
avg := pt^[0];
FOR i := 1 TO stop DO
	avg := avg + pt^[i];
END_FOR;
avg := avg / (stop + 1);

(* in a second run we calculate the variance of the array *)

array_var := (pt^[0] - avg) * (pt^[0] - avg);
FOR i := 1 TO stop DO
	array_var := array_var + (pt^[i] - avg) * (pt^[i] - avg);
END_FOR;
array_var := array_var / stop;

(* revision history
hm 	1.4.2007	rev 1.0
	function created

hm	12.12.2007	rev 1.1
	changed code for better performance
*)
END_FUNCTION

(* POU array_spr, ST *)
FUNCTION array_spr : REAL
VAR_INPUT
	pt : POINTER TO ARRAY[0..32000] OF REAL;
	size : INT;
END_VAR
VAR
	i: INT;
	stop: INT;
	array_max : REAL;
	array_min : REAL;
END_VAR

(*
version 1.0	2 oct 2006
programmer 	hugo
tested by		tobias

this function will calculate the spread of a given array.
the function needs to be called:	array_spr(adr("array"),sizeof("array"));
for example: spread of [12,0,4,1,7] is 12 - 0 = 12.
because this function works with pointers its very time efficient and it needs no extra memory.

*)
stop := (size -SIZEOF(pt)) / SIZEOF(pt);
array_min := pt^[0];
array_max := pt^[0];
FOR i := 1 TO stop DO
	IF pt^[i] > array_max THEN array_max := pt^[i];
	ELSIF pt^[i] < array_min THEN array_min := pt^[i];
	END_IF;
END_FOR;
array_spr := array_max - array_min;
END_FUNCTION

(* POU array_sum, ST *)
FUNCTION array_sum : REAL
VAR_INPUT
	pt : POINTER TO ARRAY[0..32000] OF REAL;
	size : INT;
END_VAR
VAR
	i: INT;
	stop: INT;
END_VAR


(*
version 1.0	2 oct 2006
programmer 	hugo
tested by		tobias

this function will calculate the sum of a given array.
the function needs to be called:	array_sum(adr("array"),sizeof("array"));
because this function works with pointers its very time efficient and it needs no extra memory.

*)
stop := (size -SIZEOF(pt)) / SIZEOF(pt);
array_sum := pt^[0];
FOR i := 1 TO stop DO
	array_sum := array_sum + pt^[i];
END_FOR;
END_FUNCTION

(* POU array_trend, ST *)
FUNCTION array_trend : REAL
VAR_INPUT
	pt : POINTER TO ARRAY[0..32000] OF REAL;
	size : INT;
END_VAR
VAR
	i: INT;
	stop: INT;
	x: REAL;
	stop2: INT;
END_VAR

(*
version 1.1	12 dec 2007
programmer 	hugo
tested by		tobias

this function will calculate the trend of a given array.
trend will calculate the avg of the first half of the array and then the avg of the second half, trend = avg2 - avg1.
for example:  [0,1,4,5,3,4,6,3] = 4 - 2.5 = 1.5
the function needs to be called:	array_trend(adr("array"),sizeof("array"));
because this function works with pointers its very time efficient and it needs no extra memory.

*)
stop := SHR(size,2)-1;
stop2 := SHR(stop,1);
FOR i := 0 TO stop2 DO x := x - pt^[i]; END_FOR;
IF even(stop) THEN
	FOR i := stop2 TO stop DO X := X + pt^[i]; END_FOR;
ELSE
	FOR i := stop2 + 1 TO stop DO X := X + pt^[i]; END_FOR;
END_IF;
array_trend := x / (stop2 + 1);

(* revision history
hm	2 oct 2007	rev 1.0
	original version

hm	12 dec 2007	rev 1.1
	changed code for better performance

*)
END_FUNCTION

(* POU asinH, ST *)
FUNCTION asinH : REAL
VAR_INPUT
	X : REAL;
END_VAR
VAR
END_VAR


(*
version 1.1	2 dec 2007
programmer 	hugo
tested by		tobias

this function calculates the arcus sin hyperbolicus

*)
asinH := LN(X + SQRT(X * X + 1));

(* revision history
hm		12 jan 2007	rev 1.0
	original version

hm		2. dec 2007	rev 1.1
	changed code for better performance

*)
END_FUNCTION

(* POU astro, ST *)
FUNCTION_BLOCK astro
VAR_INPUT
	m : REAL;
	AE : REAL;
	PC : REAL;
	LJ : REAL;
END_VAR
VAR_OUTPUT
	Ym : REAL;
	YAE : REAL;
	YPC : REAL;
	YLJ : REAL;
END_VAR
VAR
END_VAR

(*
version 1.0	27 mar 2007
programmer 	hugo
tested by		oscat

this function converts different length units
any unused input can simply be left open.
different inputs connected at the same time will be added up.

*)
YAE :=	AE
		+ m / 149.597870E9
		+ PC * 206265
		+ LJ * 63240;
Ym := YAE * 149.597870E9;
YPC := YAE / 206265;
YLJ := YAE / 63240;


(*
Länge Meter m SI-Basiseinheit
Astronomische Einheit* AE 1 AE = 149,597 870 · E9 m
Parsec pc 1 pc = 206265 AE = 30,857 · E15 m
Lichtjahr Lj 1 Lj = 9,460 530 · E15 m = 63240 AE = 0,306 59 pc
Ångström Å 1 Å = E–l0 m
typograph. Punkt p 1 p = 0,376 065 mm • im Druckereigewerbe
inch** in 1 in = 2,54 · E–2 m = 25,4 mm***
foot ft 1 ft = 0,3048 m = 30,48 cm
yard yd 1 yd = 0,9144 m
mile mile 1 mile = 1609,344 m
Internat. Seemeile sm 1 sm = 1852 m
Fathom fm 1 fm = 1,829 m • in der Seeschifffahrt

*)
END_FUNCTION_BLOCK

(* POU atanH, ST *)
FUNCTION atanH : REAL
VAR_INPUT
	X : REAL;
END_VAR
VAR
END_VAR


(*
version 1.1	5. jan 2008
programmer 	hugo
tested by		tobias

this function calculates the arcus tangens hyperbolicus

*)
atanH := LN((1+x)/(1-x)) * 0.5;


(* revision history
hm		12 jan 2007	rev 1.0
	original version

hm		5. jan 2008	rev 1.1
	improved code for better performance
*)
END_FUNCTION

(* POU B_TRIG, ST *)
FUNCTION_BLOCK B_TRIG
VAR_INPUT
	CLK : BOOL;
END_VAR
VAR_OUTPUT
	Q : BOOL;
END_VAR
VAR
	edge : BOOL := 0;
END_VAR

(*
version 1.0	4 aug 2006
programmer 	hugo
tested by		tobias

this block is similar to R_trig and F_trig but it generates a pulse on rising and falling edge.

executioin TIME on wago 750-841 = 5us
*)
Q := clk XOR edge;
edge := CLK;
END_FUNCTION_BLOCK

(* POU bar_graph, ST *)
FUNCTION_BLOCK bar_graph
VAR_INPUT
	X : REAL;
	rst : BOOL;
END_VAR
VAR_INPUT CONSTANT
	trigger_Low : REAL;
	trigger_High : REAL;
	Alarm_low : BOOL;
	Alarm_high : BOOL;
	log_scale : BOOL;
END_VAR
VAR_OUTPUT
	LOW, Q1, Q2, Q3, Q4, Q5, Q6, HIGH : BOOL;
	Alarm : BOOL;
	Status : BYTE;
END_VAR
VAR
	init : BOOL;
	T1, T2, T3, T4, T5 : REAL;
END_VAR
VAR_TEMP
	temp : REAL;
END_VAR

(*
	version 1.2	6 jan 2008
	programmer 	hugo
	tested BY		hans

bar graph is a muti window comparator which displays an analog input signal on 8 digital outputs.
only one output is active a any given time depending on the value of the input signal.
the output can be of linear or logarithmic scale.

*)
IF NOT init THEN
	init := TRUE;
	IF log_scale THEN
		temp := EXP(LN(Trigger_high / Trigger_low) * 0.166666666666666666666);
		T1 := trigger_low * temp;
		T2 := T1 * temp;
		T3 := T2 * temp;
		T4 := T3 * temp;
		T5 := T4 * temp;
	ELSE
		temp := (trigger_high - trigger_low) * 0.142857142;
		T1 := trigger_low + temp;
		T2 := T1 + temp;
		T3 := T2 + temp;
		T4 := T3 + temp;
		T5 := T4 + temp;
	END_IF;
END_IF;

(* clear outputs before checking *)
Q1 := FALSE;
Q2 := FALSE;
Q3 := FALSE;
Q4 := FALSE;
Q5 := FALSE;
Q6 := FALSE;
status := 110;

(* low, high and alarm can only be cleared with rst depending on alarm_low and alarm_high *)
IF NOT alarm_low THEN low := FALSE; END_IF;
IF NOT alarm_high THEN high := FALSE; END_IF;
IF rst THEN
	alarm := FALSE;
	low := FALSE;
	high := FALSE;
END_IF;

(* check and set outputs *)
IF X < trigger_low THEN
	Low := TRUE;
	status := 111;
	IF alarm_low THEN
		alarm := TRUE;
		status := 1;
	END_IF;
ELSIF X < T1 THEN
	Q1 := TRUE;
ELSIF x < t2 THEN
	Q2 := TRUE;
ELSIF x < t3 THEN
	Q3 := TRUE;
ELSIF x < T4 THEN
	Q4 := TRUE;
ELSIF x < T5 THEN
	q5 := TRUE;
ELSIF x < trigger_high THEN
	q6 := TRUE;
ELSE
	high := TRUE;
	status := 112;
	IF alarm_high THEN
		alarm := TRUE;
		status := 2;
	END_IF;
END_IF;

(* revision history
hm	22. feb 2007	rev 1.0
	original version

hm	2. dec 2007		rev 1.1
	chaged code for better performance

hm	6. jan 2008		rev 1.2
	further performance improvement

*)
END_FUNCTION_BLOCK

(* POU BCD_TO_INT, ST *)
FUNCTION BCD_TO_INT : INT
VAR_INPUT
	in : BYTE;
END_VAR
VAR
END_VAR

(*
version 1.0	13 dec 2007
programmer 	hugo
tested by		tobias

this function converts a two digit bcd number into an integer.
*)
	BCD_TO_INT := (in AND 16#0F) + (SHR(in,4) * 10);

(* revision history
hm	13.12.2007
	original version

*)
END_FUNCTION

(* POU Bit_Count, ST *)
FUNCTION Bit_Count : INT
VAR_INPUT
	IN : DWORD;
END_VAR
VAR
END_VAR

(*
version 1.1	10 sep 2007
programmer 	hugo
tested by		tobias

BIT_COUNT counts the amount True of bits in a dword.
for exabple: bit_count(3) returns 2 because two bits (bits 0 and 1) are true and all others are false. 

*)
WHILE in > 0 DO
	IF in.0 THEN Bit_Count := Bit_Count +1; END_IF;
	in := SHR(in,1);
END_WHILE;

(* revision history
5.7.2007	rev 1.0		original version

10.9.2007	rev 1.1		hm
	changed algorithm for better performace
	the execution time has reduced by a factor of 5
	deleted unused variable temp
*)
END_FUNCTION

(* POU Bit_of_Dword, ST *)
FUNCTION Bit_of_Dword : BOOL
VAR_INPUT
	in : DWORD;
	N : BYTE;
END_VAR
VAR
	temp: DWORD;
END_VAR

(*
version 1.0	4 aug 2006
programmer 	hugo
tested by		tobias

this function extracts a single bit from the nth position from right (right is lowest bit)
the lowest Bit (Bit0 from in) is selected with N=0.
 *)
temp := SHR(in,n);
Bit_of_Dword := temp.0;
END_FUNCTION

(* POU blind_actuator, ST *)
 FUNCTION_BLOCK blind_actuator
VAR_INPUT
	UP, DN : BOOL;
	S_IN : BYTE;
	T_UD : TIME := T#10s;
	T_Angle : TIME := T#3s;
END_VAR
VAR_INPUT CONSTANT
	T_lockout : TIME := t#100ms;
END_VAR
VAR_OUTPUT
	pos, ang : BYTE;
	QU, QD : BOOL;
	status : BYTE;
END_VAR
VAR
	position, angle : rmp_B;
	lock : interlock;
END_VAR

(*
version 1.1	6 oct 2007
programmer 	hugo
tested by		tobias

blind actuator drives the up and down motor of a blind. T_lockout specifies the time between up or dn becomes active. 
To change direction there must be a minimum wait time to allow the motors to come to rest first.
the up and down outputs QU and QD are controlled by the inputs UP and DN.
the outputs pos and ang simulate the position of the blind pos = 0 means blind is down and pos = 255 = blind is up.
the angle 0 means vertical posisition of the slates and 255 means horizontal position of the slates.


*)
(* make sure only one motor is active at a given time *)
lock(i1 := UP, I2 := DN, TL := T_lockout);

(* ramp up or down to simulate the angle position of the blind slats *)
angle(en := lock.Q1 OR lock.Q2, UP := lock.Q1, PT := T_Angle);
position(en := lock.Q1 AND angle.high OR lock.Q2 AND angle.low, up := lock.Q1, PT := T_UD);

(* set the outputs *)
pos := position.Out;
ang := angle.Out;
QU := lock.Q1;
QD := lock.Q2;

(* set the status output *)
IF UP AND DN THEN
	IF s_in < 10 AND S_in > 1 THEN status := s_in; ELSE status := 1; END_IF;			(* error up and down together are not allowed *)
ELSIF S_IN > 0 THEN
	status := S_IN;
ELSIF UP THEN
	status := 101;
ELSIF DN THEN
	status := 102;
ELSE
	status := 0;
END_IF;


(* revision history
hm	29. sep 2007	rev 1.0
	original release

hm	6. oct 2007		rev 1.1
	rearranged outputs
	
*)
END_FUNCTION_BLOCK

(* POU rmp_B, ST *)
FUNCTION_BLOCK rmp_B
VAR_INPUT
	SET : BOOL := FALSE;
	PT : TIME;
	EN : BOOL := TRUE;
	UP : BOOL := TRUE;
	RST : BOOL := FALSE;
END_VAR
VAR_OUTPUT
	out : BYTE;
	busy: BOOL;
	high : BOOL;
	low : BOOL;
END_VAR
VAR
	last_step : DWORD;
	now : DWORD;
	tmp: DWORD;
	edge: BOOL;
	N : BYTE;
	init: BOOL;
END_VAR

(*
	version 1.6	25 dec 2007
	programmer 	oscat
	tested BY		oscat

this ramp generator generates a byte wide ramp with 255 steps
the generator has an asynchronous set and reset
the ramp is controlled by PT which is the total ramp time for a full sweep from 0..255
an UD input controlls the direction Up or Down and the E input enables the ramp generation
a busy output indicates that the ramp is running, busy false means output is stable.
the outputs low and high will be true when the output has reached its max or min value.

*)
(* read system time *)
now := T_PLC_MS();

(* init code for startup *)
IF NOT init THEN
	init := TRUE;
	last_step := now;
END_IF;

(* calculate the necessary step response *)
IF pt = t#0s THEN
	tmp := 255;
ELSE
	tmp := SHL(now - last_step, 8) / (TIME_TO_DWORD(pt));
END_IF;
IF tmp > 255 THEN N:= 255; ELSE N:= DWORD_TO_BYTE(tmp); END_IF;

(* detetct edge on en *)
IF en AND NOT edge THEN
	last_step := now;
(* check for asynchronous set or reset *)
ELSIF rst THEN
	out := 0;
ELSIF set  THEN
	out := 255;
ELSIF en AND N > 0 THEN
	(* generate ramp *)
	last_step := now;
	IF UP THEN
		IF out > 255 - N THEN out := 255; ELSE out := out + N; END_IF;
	ELSE
		IF out < N THEN out := 0; ELSE out := out - N; END_IF;
	END_IF;
END_IF;
edge := en;

(* checks for outputs stable and reset or set busy flag *)
IF out = 0 THEN
	busy := FALSE;
	low := TRUE;
	high := FALSE;
ELSIF out = 255 THEN
	busy := FALSE;
	high := TRUE;
	low := FALSE;
ELSE
	busy := en;
	high := FALSE;
	low := FALSE;
END_IF;


(* revision history

hm 5.10.2006	rev 1.1
	added busy output
hm 17.1.2007	rev 1.2
	renamed input ud to up for better usability
	deleted unused variable step

hm	17.9.2007	rev 1.3
	replaced time() with t_plc_ms() for compatibility reasons

hm	28. sep 2007	rev 1.4
	added outputs on and off
	busy is now disabled while en is false
	new coding for higher accuracy and performance

hm	5. oct 2007		rev 1.5
	added statements to allow for PT to be t#0s output jumps to max or min immediately

hm	25. dec 2007	REV 1.6
	IMPROOVED CODE FOR BETTER PERFORMANCE
*)
END_FUNCTION_BLOCK

(* POU interlock, ST *)
FUNCTION_BLOCK interlock
VAR_INPUT
	I1, I2 : BOOL;
	TL : TIME;
END_VAR
VAR_OUTPUT
	Q1, Q2 : BOOL;
END_VAR
VAR
	T1, T2 : TOF;
END_VAR

(*
version 1.0	28 sep 2007
programmer 	hugo
tested by		tobias

INTERLOCK has two inputs I1 and I2 which drive the corresponding outputs Q1 and Q2.
the inputs signals lock each other out and therfore I1 can only drive Q1 when I2 is Low and vice versa.
The input TL specifies a dead time between two outputs can become active.
an output can only become active when the other output was not active for the time TL.

*)
(* the input signal have a run delay to lockout the other input *)
T1(IN := I1, PT := TL);
T2(IN := I2, PT := TL);

Q1 := I1 AND NOT t2.Q;
Q2 := I2 AND NOT t1.Q;


(* revision history

hm	28 sep 2007		rev 1.0
	original version

*)
END_FUNCTION_BLOCK

(* POU blind_control, ST *)
FUNCTION_BLOCK blind_control
VAR_INPUT
	UP, DN : BOOL;
	S_IN : BYTE;
	pi : BYTE;
	ai : BYTE;
	T_UD, T_ANGLE : TIME;
END_VAR
VAR_INPUT CONSTANT
	sens : BYTE := 5;
	T_Lockout: TIME := T#100ms;
END_VAR
VAR_OUTPUT
	pos, ang : BYTE;
	MU, MD : BOOL;
	status : BYTE;
END_VAR
VAR
	act : blind_actuator;
	delta : BYTE;
END_VAR

(*
version 1.3	30. oct 2007
programmer 	hugo
tested by		tobias


*)
IF UP AND DN THEN
	(* automatic modus detected *)
	(* first find correct position *)
	IF BYTE_TO_INT(act.pos) < BYTE_TO_INT(pi) - delta THEN
		act.UP := TRUE;
		act.DN := FALSE;
		delta := 0;
		act.S_IN := 121;
	ELSIF BYTE_TO_INT(act.pos) > BYTE_TO_INT(pi) + delta THEN
		act.UP := FALSE;
		act.DN := TRUE;
		delta := 0;
		act.S_IN := 122;
	(* regulate angle *)
	ELSIF BYTE_TO_INT(act.ang) < BYTE_TO_INT(ai) - delta AND T_angle > T#100ms THEN
		act.UP := TRUE;
		act.DN := FALSE;
		delta := 0;
		act.S_IN := 123;
	ELSIF BYTE_TO_INT(act.ang) > BYTE_TO_INT(ai) + delta AND T_angle > T#100ms THEN
		act.UP := FALSE;
		act.DN := TRUE;
		delta := 0;
		act.S_IN := 124;
	(* correct position reached *)
	ELSE
		act.UP := FALSE;
		act.DN := FALSE;
		delta := sens;
		act.S_IN := 0;
	END_IF;
ELSE
	act.UP := UP;
	act.DN := DN;
END_IF;

(* hand over status *)
IF s_in > 0 THEN act.S_IN := S_IN; END_IF;

(* blind control calls blind_actuator *)
act(T_UD:=T_UD, T_ANGLE:=T_ANGLE, T_lockout := T_Lockout);
pos := act.pos;
ang := act.ang;
MU := act.QU;
md := act.QD;
status := act.status;

(* revision history
hm	29. sep 2007	rev 1.0
	original release

hm	6. oct 2007		rev 1.1
	rearranged outputs
	integrated blind_actuator into blind_control

hm	16. oct 2007	rev 1.2
	ignore angle when t_angle = 0

hm 29. oct 2007	rev 1.3
	added lockout configuration time for motor direction change
	sens has a setup value of 5
*)
END_FUNCTION_BLOCK

(* POU blind_input, ST *)
FUNCTION_BLOCK blind_input
VAR_INPUT
	pos, ang : BYTE;
	S1, S2 : BOOL;
	in : BOOL;
	pi, ai : BYTE;
END_VAR
VAR_INPUT CONSTANT
	single_switch : BOOL := FALSE;
	click_mode : BOOL := TRUE;
	click_time : TIME := T#200ms;
	click_timeout : TIME := T#60s;
	manual_timeout: TIME := T#1h;
END_VAR
VAR_OUTPUT
	QU, QD : BOOL;
	status : BYTE;
	po, ao : BYTE;
END_VAR
VAR
	click_run : TOF;
	tog1, tog2 : TOGGLE;
	pl1, pl2 : Pulse_Length;
	SU, SD : BOOL;
	last_act: DWORD;
	tx: DWORD;
END_VAR

(*
version 1.2	30 dec 2007
programmer 	hugo
tested by		tobias


*)
(* read system_time *)
tx := T_PLC_MS();

(* single or double switch operation *)
IF click_mode THEN
	PL1(in := S1, T_short := click_time, T_long := click_time);
	PL2(in := S2, T_short := click_time, T_long := click_time);
	(* a timeout needs to be added for click enable *)
	click_run(IN := pl1.short OR pl2.short, PT := click_timeout);
	tog1(clk := pl1.short, rst := pl1.long OR pl2.short OR pl2.long OR NOT click_run.Q);
	tog2(clk := pl2.short, rst := pl2.long OR pl1.short OR pl1.long OR NOT click_run.Q);

	SU := tog1.Q OR PL1.long;
	SD := tog2.Q OR pl2.long;
ELSE
	tog1(CLK := NOT S1);
	SU := (S1 AND NOT tog1.Q AND single_switch) OR (NOT single_switch AND S1);
	SD := (S1 AND tog1.Q AND single_switch) OR (NOT single_switch AND S2);
END_IF;

(* Forced Input is active *)
IF in THEN
	QU := TRUE;
	QD := TRUE;
	po := pi;
	ao := ai;
	status := 131;

(* in manual mode set ps and as to actual values *)
ELSIF SU OR SD THEN
	po := pos;
	ao := ang;
	last_act := tx;
	QU := SU;
	QD := SD;
	IF su THEN status := 132; ELSE status := 133; END_IF;

(* enable automatik mode after auto timer has expired *)
ELSIF manual_timeout > t#0s AND tx - last_act >= TIME_TO_DWORD(manual_timeout) THEN
	QU := TRUE;
	QD := TRUE;
	status := 134;

(* no input active *)
ELSE
	QU := FALSE;
	QD := FALSE;
	status := 0;
END_IF;


(* revision history
hm	29. sep 2007	rev 1.0
	original release

hm	6. oct 2007		rev 1.1
	renamed ps and as to po and ao

hm	30. dec 2007	rev 1.2
	added click_timeout variable and function

*)
END_FUNCTION_BLOCK

(* POU TOGGLE, ST *)
FUNCTION_BLOCK TOGGLE
VAR_INPUT
	CLK : BOOL;
	rst : BOOL := FALSE;
END_VAR
VAR_OUTPUT
	Q : BOOL;
END_VAR
VAR
	edge : BOOL;
END_VAR

(*
version 1.0	13 sep 2007
programmer 	hugo
tested by		tobias

toggle flip flop the output changes state with every rising edge of clk.

*)
IF rst THEN
	q := 0;
ELSIF clk AND NOT edge THEN
	Q := NOT Q;
END_IF;
edge := clk;

(* revision history

hm	13.9.2007		rev 1.0
	original version

*)
END_FUNCTION_BLOCK

(* POU Pulse_Length, ST *)
FUNCTION_BLOCK Pulse_Length
VAR_INPUT
	in : BOOL;
END_VAR
VAR_OUTPUT
	short : BOOL;
	middle : BOOL;
	long : BOOL;
END_VAR
VAR_INPUT CONSTANT
	T_short : TIME := t#100ms;
	T_long : TIME := t#1s;
END_VAR
VAR
	tx : TIME;
	tn: TIME;
	edge : BOOL;
END_VAR

(*
version 1.1	15 sep 2007
programmer 	oscat
tested by		tobias

Pulse_length indicates on 3 outputs if an input pulse had been shorter than T_short (short = True), longer than T_long (long = True) or between T_short and T_long (middle = True).

*)
(* read system time *)
tx := DWORD_TO_TIME(T_PLC_MS());

(* reset outputs, they should only be active 1 cycle *)
short := FALSE;
Middle := FALSE;
long := FALSE;

(* detect rising edge *)
IF in AND NOT edge THEN
	edge := TRUE;
	tn := tx;

(* detect for falling edge *)
ELSIF NOT in AND edge THEN
	edge := FALSE;
	tn := tx - tn;
	IF tn < t_short THEN
		short := TRUE;
	ELSIF tn > t_long THEN
		long := TRUE;
	ELSE
		Middle := TRUE;
	END_IF;

(* generate long pulse as soon as T_long is reached *)
ELSIF in AND tx - tn > t_long THEN
	long := TRUE;
END_IF;


(* revision history

hm	15. feb 2006	rev 1.0
	original version

hm	15 sep 2007		rev 1.1
	replaced Time() with T_PLC_MS for compatibility and performance reasons

*)
END_FUNCTION_BLOCK

(* POU blind_night, ST *)
FUNCTION_BLOCK blind_night
VAR_INPUT
	UP, DN : BOOL;
	S_IN : BYTE;
	pi, ai : BYTE;
	E_night : BOOL := TRUE;
	E_day	: BOOL := TRUE;
	dtin : DT;
	sunrise, sunset : TOD;
END_VAR
VAR_INPUT CONSTANT
	sunrise_offset : TIME;
	sunset_offset : TIME;
	night_position : BYTE := 0;
	night_angle : BYTE := 0;
END_VAR
VAR_OUTPUT
	QU, QD : BOOL;
	status : BYTE;
	po, ao : BYTE;
END_VAR
VAR
	night : BOOL;
	last_night, last_day : DATE;
END_VAR

(*
version 1.2	6 oct 2007
programmer 	hugo
tested by		tobias


*)
IF NOT (up AND dn) AND night THEN
	(* manual operation at night will cancel operation for one night *)
	night := FALSE;
ELSIF (DT_TO_TOD(dtin) > sunset + sunset_offset) AND (last_night < DT_TO_DATE(dtin)) AND NOT night AND e_night THEN
	(* enable night *)
	night := TRUE;
	last_night := DT_TO_DATE(dtin);
ELSIF (DT_TO_TOD(dtin) > sunrise + sunrise_offset) AND (last_day < DT_TO_DATE(dtin)) AND night AND e_day AND (last_night < DT_TO_DATE(dtin)) THEN
	(* disable night *)
	night := FALSE;
	last_day := DT_TO_DATE(dtin);
END_IF;

(* shade at night only in auto mode and enable = true *)
IF UP AND DN AND night THEN
	status := 141;
	po := night_position;
	ao := night_angle;
ELSE
	QU := UP;
	QD := DN;
	po := pi;
	ao := ai;
	status := s_in;
END_IF;


(* revision history
hm	29. sep 2007	rev 1.0
	original version

hm	5. oct 2007		rev 1.1
	added enable input

hm	6. oct 2007		rev 1.2
	added pos and angle inputs and outputs
	night position and angle can now be configured
	any manual operation at night will cancel night operation

*)
END_FUNCTION_BLOCK

(* POU blind_scene, ST *)
FUNCTION_BLOCK blind_scene
VAR_INPUT
	UP, DN : BOOL;
	S_IN : BYTE;
	pi, ai : BYTE;
	enable : BOOL;
	swrite : BOOL;
	scene : BYTE;
END_VAR
VAR_INPUT CONSTANT
END_VAR
VAR_OUTPUT
	QU, QD : BOOL;
	status : BYTE;
	po, ao : BYTE;
END_VAR
VAR RETAIN
	sx : ARRAY[0..15,0..2] OF BYTE;
END_VAR
VAR_TEMP
	x : BYTE;

END_VAR

(*
version 1.1	29. jan 2008
programmer 	hugo
tested by		tobias


*)
(* delete all bits except the lower 4 of scene *)
x := scene AND 16#0F;

IF enable AND sx[x,2] > 0 AND UP AND DN THEN
	po := sx[x,0];
	ao := sx[x,1];
	status := 160 + x;  (* Status number is 160 to 175 for the 16 scenes *)
	QU := TRUE;
	QD := TRUE;
ELSE
	QU := UP;
	QD := DN;
	status := S_IN;
	po := pi;
	ao := ai;
END_IF;

(* write scene if necessary *)
IF swrite THEN
	status := 176;		(* write scene *)
	sx[x,0] := pi;
	sx[x,1] := ai;
	IF enable THEN sx[x,2] := 1; ELSE sx[x,2] := 0; END_IF; (* if sx[x,2] = 0 the scene is disabled *)
END_IF;


(* revision history
hm	24. oct 2007	rev 1.0
	original release

hm		29.1.2008	rev 1.1
	replaced shr/shl with and for better performance
*)
END_FUNCTION_BLOCK

(* POU blind_security, ST *)
FUNCTION_BLOCK blind_security
VAR_INPUT
	UP, DN : BOOL;
	S_IN : BYTE;
	pi, ai : BYTE;
	FIRE : BOOL;
	Wind : BOOL;
	Alarm : BOOL;
	Door : BOOL;
	Rain : BOOL;
END_VAR
VAR_INPUT CONSTANT
	Alarm_UP : BOOL := TRUE;
END_VAR
VAR_OUTPUT
	QU, QD : BOOL;
	status : BYTE;
	po, ao : BYTE;
END_VAR
VAR
END_VAR

(*
version 1.1	6. oct 2007
programmer 	hugo
tested by		tobias


*)
IF Fire THEN
	QU := TRUE;
	QD := FALSE;
	status := 111;
ELSIF Wind THEN
	QU := TRUE;
	QD := FALSE;
	status := 112;
ELSIF alarm THEN
	QU := Alarm_up;
	QD := NOT Alarm_up;
	status := 113;
ELSIF Door THEN
	QU := TRUE;
	QD := FALSE;
	status := 114;
ELSIF Rain AND NOT (up XOR dn) THEN
	QU := FALSE;
	QD := TRUE;
	status := 115;
ELSE
	QU := UP;
	QD := DN;
	status := S_IN;
	po := pi;
	ao := ai;
END_IF;


(* revision history
hm	29. sep 2007	rev 1.0
	original release

hm	6. oct 2007		rev 1.1
	added pos and angle inputs and outputs
	manual will override rain position
	alarm position can now be configured

*)
END_FUNCTION_BLOCK

(* POU BLIND_SHADE, ST *)
FUNCTION_BLOCK BLIND_SHADE
VAR_INPUT
	UP, DN : BOOL;
	S_IN : BYTE;
	pi, ai : BYTE;
	enable : BOOL;
	sun : BOOL;
	dtin : DT;
	sunrise, sunset : TOD;
	sun_hor, sun_ver : REAL;
END_VAR
VAR_INPUT CONSTANT
	sunrise_offset : TIME := T#1h;
	sunset_preset : TIME := T#1h;
	direction : REAL := 180;
	angle_offset : REAL := 80;
	slat_width : REAL := 80;
	Slat_spacing : REAL := 60;
	Shade_delay : TIME := T#60s;
END_VAR
VAR_OUTPUT
	QU, QD : BOOL;
	status : BYTE;
	po, ao : BYTE;
END_VAR
VAR
	angle: REAL;
	sun_delay : TOF;
END_VAR

(*
version 1.2	24 nov 2007
programmer 	hugo
tested by		tobias


*)
(* the input sun is sent through tof which will delay the shade for the time shade_delay *)
sun_delay(IN := sun, PT := shade_delay);

IF UP AND DN AND enable AND sun_delay.Q AND sun_hor > direction - angle_offset AND sun_hor < direction + angle_offset AND
	DT_TO_TOD(dtin) > sunrise + sunrise_offset AND DT_TO_TOD(dtin) < sunset - sunset_preset THEN
	status := 151;
	QU := UP;
	QD := DN;
	(* position is fully down *)
	po := 0;
	(* shading is active now calculate the slat angle *)
	(* calculate the max angle for the blind *)
	angle := deg(ATAN(slat_spacing / slat_width));
	(* check if sun angle is between 0 and max angle *)
	IF sun_ver > 0 AND sun_ver < angle THEN
		angle := sun_ver + deg(ACOS(COS(Rad(sun_ver))*slat_spacing / Slat_width));
		ao := INT_TO_BYTE(LIMIT(0,TRUNC(angle * 255 / 90), 255));
	ELSE
		ao := 255;
	END_IF;
ELSE
	QU := UP;
	QD := DN;
	po := pi;
	ao := ai;
	status := S_IN;
END_IF;

(* revision history
hm	15 oct. 2007	rev 1.0
	original version

hm	19. oct 2007	rev 1.1
	manual mode was not detected because outputs were checked and not inputs UP and DN

hm	24. nov 2007	rev 1.2
	added shade_delay to avoid constant up and down if sun is out parcially
*)
END_FUNCTION_BLOCK

(* POU deg, ST *)
FUNCTION deg : REAL
VAR_INPUT
	rad : REAL;
END_VAR
VAR
END_VAR
VAR
END_VAR

(*
version 1.1	16 oct 2007
programmer 	hugo
tested by		tobias

this function converts degrees into Radiant
execution time on wago 750 - 841 =  10  us
*)
deg := modR(57.29577951308232 * Rad, 360);

(* revision history
hm	4. aug 2006		rev 1.0
	original version

hm 	16. oct 2007	rev 1.1
	added modr statement which prohibits deg to become bigger than 360

*)
END_FUNCTION

(* POU Rad, ST *)
FUNCTION Rad : REAL
VAR_INPUT
	deg : REAL;
END_VAR
VAR
END_VAR

(*
version 1.0	4 aug 2006
programmer 	hugo
tested by	tobias

this function converts Radiant to degrees

*)
Rad := modR(0.0174532925199433 * deg,PI2);

(* revision history
hm	4. aug 2006
	original version

hm 	16. oct 2007
	added modr statement which prohibits rad to become bigger than 2PI

*)
END_FUNCTION

(* POU modR, ST *)
FUNCTION modR : REAL
VAR_INPUT
	in : REAL;
	divi : REAL;
END_VAR

VAR
END_VAR

(*
version 1.1	4 aug 2006
programmer 	hugo
tested by		tobias

this is a modulo funtion for real numbers
modr(5.5,2.5) = 0.5


execution time on wago 750 - 841 =  29  us
*)
IF divi = 0 THEN
	modR := 0;
ELSE
	modR := in - TRUNC(in / divi) * divi;
END_IF;

(* revision history

hm 4.8.2006	rev 1.0

hm 28.1.2007	rev 1.1
	modr(x,0) will deliver the result 0

*)
END_FUNCTION

(* POU Boiler, ST *)
FUNCTION_BLOCK Boiler
VAR_INPUT
	T_upper : REAL;
	T_lower : REAL;
	Pressure : BOOL := TRUE;
	enable : BOOL := TRUE;
	Req_1 : BOOL;
	Req_2 : BOOL;
	Boost : BOOL;
END_VAR
VAR_INPUT CONSTANT
	t_upper_min : REAL := 50;
	t_upper_max : REAL := 60;
	T_lower_enable : BOOL;
	T_lower_max : REAL := 60;
	T_request_1 : REAL := 70;
	T_request_2 : REAL := 50;
	T_request_hys : REAL := 5;
	T_protect_high : REAL := 80;
	T_protect_low : REAL := 10;
END_VAR
VAR_OUTPUT
	Heat : BOOL;
	error : BOOL;
	status : BYTE;
END_VAR
VAR
	edge: BOOL;
	boost_mode: BOOL;
	flag_0 : BOOL;
	flag_1: BOOL;
	flag_2: BOOL;
END_VAR

(*
version 1.0	27 feb 2007
programmer 	hugo
tested by		tobias

this function block controls a hot water boiler. The Boiler can be equipped with two temperature sensors on top and bottom of the tank, T_LOWER_ENABLE must be set to True in this case.
alternatively can BOILER be configured for one (TOP) temperature sensor only (T_LOWER_ENABLE set to False).
A Pressure sensor is used to detect fresh water pressure and disable all heating if there is no water pressure. This input is dset to True by default, so if it is not used it can simply be left open.
A enable input enables the hot water heating while it is set to True. alternatively can a Ture on Req_1 or Req_2 start the heating to predefined temperatures during setup.
A low to high edge on the boost input will start heating imediately until T_upper_max is reached, it can be used to generate extra hot water when needed.

*)
(* read sensors and check for valid data *)
IF t_upper > t_protect_high THEN
	status := 1;
	heat := FALSE;
	error := TRUE;
ELSIF t_upper < t_protect_low THEN
	status := 2;
	heat := TRUE;
	error := TRUE;
ELSIF t_lower > T_protect_high AND t_lower_enable THEN
	status := 3;
	heat := FALSE;
	error := TRUE;
ELSIF t_lower < t_protect_low AND t_lower_enable THEN
	status := 4;
	heat := TRUE;
	error := TRUE;
ELSIF NOT pressure THEN
	status := 5;
	heat := FALSE;
	error := TRUE;
ELSIF req_1 OR req_2 OR enable OR boost THEN
	error := FALSE;

	(* determine if heat needs to be turned on *)
	IF boost AND NOT edge AND t_upper < t_upper_max THEN
		status := 101;
		heat := TRUE;
		boost_mode := TRUE;
	ELSIF enable AND t_upper < T_upper_min THEN
		status := 102;
		heat := TRUE;
	ELSIF req_1 AND t_upper < T_request_1 THEN
		status := 103;
		heat := TRUE;
	ELSIF req_2 AND t_upper < t_request_2 THEN
		status := 104;
		heat := TRUE;
	END_IF;

	(* determine the shut off temperature *)
	IF heat THEN
		IF (enable OR boost_mode) THEN
			flag_0 := TRUE;
			IF T_lower_enable AND T_lower > T_lower_max THEN
				flag_0 := FALSE;
				boost_mode := FALSE;
			ELSIF NOT T_lower_enable AND T_upper > T_upper_max THEN
				flag_0 := FALSE;
				boost_mode := FALSE;
			END_IF;
		ELSE
			flag_0 := FALSE;
		END_IF;
		IF req_1 AND T_upper > T_request_1 + T_request_hys THEN flag_1 := FALSE; ELSE flag_1 := req_1; END_IF;
		IF req_2 AND T_upper > T_request_2 + T_request_hys THEN flag_2 := FALSE; ELSE flag_2 := req_2; END_IF;

		(* shut off heat if no longer needed *)
		heat := flag_0 OR flag_1 OR flag_2;
		IF heat = FALSE THEN status := 100; END_IF;
	END_IF;
ELSE
	status := 100;
	heat := FALSE;
	error := FALSE;
END_IF;
edge := boost;
END_FUNCTION_BLOCK

(* POU pressure, ST *)
FUNCTION_BLOCK pressure
VAR_INPUT
	mws : REAL;
	torr : REAL;
	att : REAL;
	atm : REAL;
	pa : REAL;
	bar : REAL;
END_VAR
VAR_OUTPUT
	Ymws : REAL;
	Ytorr : REAL;
	Yatt : REAL;
	Yatm : REAL;
	Ypa : REAL;
	Ybar : REAL;
END_VAR
VAR
END_VAR

(*
version 1.0	27 mar 2007
programmer 	hugo
tested by		oscat

this function converts different pressure units
any unused input can simply be left open.
different inputs connected at the same time will be added up.
*)
Ybar := bar +
		pa / 100000 +
		0.980665 * att +
		1.01325 * atm +
		0.001333224 * torr +
		0.0980665 * mws;
Ymws := ybar / 0.0980665;
Ytorr := ybar / 0.001333224;
Yatt := ybar / 0.980665;
yatm := ybar / 1.01325;
Ypa := ybar * 100000;


(*
Druck, Pascal Pa 1 Pa = 1 N/m2 = 1 kg/(s2 �E m) . 0,75 �E 10.2 mmHg
mechanische 1 MPa = 1 N/mm2 . fur Festigkeitsangaben
Spannung Bar bar 1 bar = 105 Pa = 103 mbar = 105 kg/(s2 �E m)
Millimeter- mmHg 1 mmHg = 133,322 Pa = 1,333 22 mbar
Quecksilbersaule . nur in Heilkunde zulassig
physik. Atmosphare atm 1 atm = 1,013 25 bar
techn. Atmosphare at 1 at = 1 kp/cm2 = 0,980665 bar
Torr Torr 1 Torr = (101325/760) Pa = 1,333224 mbar
Meter-Wassersaule mWS 1 mWS = 9806,65 Pa = 98,0665 mbar
psi lbf/in2 1 lbf/in2 = 68,947 57 mbar = 6894,757 Pa

*)
END_FUNCTION_BLOCK

(* POU Burner, ST *)
FUNCTION_BLOCK Burner
VAR_INPUT
	in : BOOL;
	stage2 : BOOL;
	over_temp : BOOL;
	oil_temp : BOOL := TRUE;
	Flame : BOOL;
	rst : BOOL;
	rst_timer : BOOL;
END_VAR
VAR_INPUT CONSTANT
	pre_heat_time : TIME := t#5s;
	pre_vent_time : TIME := t#15s;
	pre_ignite_time : TIME := t#5s;
	post_ignite_time : TIME := t#25s;
	stage2_delay : TIME := t#10s;
	safety_time : TIME := t#5s;
	lockout_time : TIME := t#10s;
	multiple_ignition : BOOL := TRUE;
	KW1 : REAL;
	KW2 : REAL;
END_VAR
VAR_OUTPUT
	motor : BOOL;
	coil1 : BOOL;
	coil2 : BOOL;
	pre_heat: BOOL;
	ignite : BOOL;
	runtime1 : REAL;
	runtime2 : REAL;
	KWh : REAL;
	cycles : REAL;
	status : BYTE;
	fail : BOOL;
END_VAR
VAR
	state : BYTE;
	last : TIME;
	tx: TIME;
	last_change: TIME;
	timer1 : ontime;
	timer2 : ontime;
	oil_temp_last: BOOL;
END_VAR

(*
version 1.5	15 sep 2007
programmer 	oscat
tested by		tobias

burner ist eine Oel-Brenner_steuerung fuer nichtmodulierende Oelbrenner
die steuerung kann ueber setup werte programmiert werden und entsprechenden brennern angepasst werden.
die vorheizzeit ist die zeit die eine oelvorwaermung aufgeheizt wird bevor der motor gestartet wird.
der eingang oil_temp gibt an ob die oil_temp erreicht wurde, er ist default auf true und kann auch offen gelassen werden.
die vorbelueftungszeit ist die zeit die der luefter laeuft bevor die oelzufuhr freigegeben wird.
die vorzuendzeit iust diejenige zeit die die zuendung vor offnen des oelventiel gestartet wird.
nachzuendzeit ist die zeit die nach entzuendung der flamme noch gezuendet wird.
die sicherheitszeit ist die zeit nach der die oelzufuhr gesperrt wird wenn keine flamme entsteht.
nach ablauf der sicherheitszeit wird ein fehler flag gesetzt und kann erst nach der sperrzeit wieder durch einen reset geloescht werden.
waehrend der sperrzeit ist keine weitere zuendung oder einschalten moeglich.
das flag mehrfachzuendung gibt an ob eine erloschene flamme in betrieb automatisch wieder gezuendet werden soll.
der flammwaechster liegt auf eingang flamme, ein uebertemperaturschutz auf dem eingang over_temp
der betriebsstundenzaehler gibt die brennerstunden in stunden als real ausgabewer an.
der ausgang motor steuert den luefter / pumpenmotor, oil_ventil schaltet das oil ventil und zuendung schaltet die zuendung ein.

if output fail > 0 an error happened and the output has an error code:
0 :	no error
1 :	pre heating time expired and oil temp input is not true
2 :	flame monitor is active during preheating time
3 :	flame monitor active during pre_ventilation_time
4 :	no ignoition during safety time
5 :	no flame during operation
9 :	overtemp input is true

*)
(* read system time *)
tx := DWORD_TO_TIME(T_PLC_MS());

(* check rst input and overtemp *)
IF rst OR over_temp OR state = 0 THEN
	IF status > 0 AND tx - last_change >= lockout_time AND rst THEN
		status := 110;
		fail := FALSE;
		state := 1;
	ELSE
		(* normaler reset *)
		motor := FALSE;
		coil1 := FALSE;
		coil2 := FALSE;
		ignite := FALSE;
		pre_heat := FALSE;
		IF over_temp THEN
			status := 9;
			fail := TRUE;
		END_IF;
		last_change := tx;
		last := tx;
		state := 1;
	END_IF;
END_IF;

(* check for timer rst and rst timer if true *)
IF rst_timer THEN
	timer1( rst := TRUE);
	timer1.rst := FALSE;
	timer2(rst := TRUE);
	timer2.rst := FALSE;
END_IF;

(* quit here if an error is present *)
IF (status > 0 AND status < 100) OR rst THEN RETURN; END_IF;

(* start sequence *)
CASE state OF

1:	(* in signal starts oil pre heating *)
	IF in AND flame THEN
		state := 7;
		pre_heat := FALSE;
		status := 2;
		last_change := tx;
	ELSIF in THEN
		pre_heat := TRUE;
		state := 2;
		last_change := tx;
	END_IF;

2:	(* after pre_heating time start motor *)
	IF (tx- last_change >= pre_heat_time AND oil_temp) OR (oil_temp AND NOT oil_temp_last) THEN
		motor := TRUE;
		state := 3;
		last_change := tx;
	(* pre_heat_time ist abgelaufen und oil_temp ist nicht aktiv *)
	ELSIF tx - last_change >= pre_heat_time AND NOT oil_temp THEN
		state := 7;
		pre_heat := FALSE;
		status := 1;
		last_change := tx;
	(* flame monitor cannot be active at this time *)
	ELSIF flame THEN
		state := 7;
		pre_heat := FALSE;
		status := 2;
		last_change := tx;
	END_IF;

3:	(* abwarten bis zündung eingeschaltet werden kann *)
	IF tx - last_change >= pre_vent_time - pre_ignite_time THEN
		ignite := TRUE;
		state := 4;
		last_change := tx;
	(* flame monitor cannot be active at this time *)
	ELSIF flame THEN
		state := 7;
		pre_heat := FALSE;
		motor := FALSE;
		status := 3;
		last_change := tx;
	END_IF;

4:	(* warten bis oelzufuhr geoeffnet werden darf *)
	IF tx - last_change >= pre_ignite_time THEN
		coil1 := TRUE;
		state := 5;
		last_change := tx;
	END_IF;

5:	(* warten auf flammwaechter und falls noetig abschalten *)
	IF tx - last_change >= safety_time OR flame THEN
		IF NOT flame THEN
			(* notabschaltung da flammwaechster nicht angesprochen hat *)
			state := 7;
			motor := FALSE;
			coil1 := FALSE;
			pre_heat := FALSE;
			ignite := FALSE;
			status := 4;
			last_change := tx;
		ELSE
			state := 6;
			last_change := tx;
		END_IF;
	END_IF;

6:	(* brenner läuft, flammueberwachung und nach ablauf der nachigniteszeit ignite abschalten *)
	IF NOT flame AND NOT multiple_ignition THEN
		(* notabschaltung da flammwaechster keine flamme meldet *)
		state := 7;
		motor := FALSE;
		coil1 := FALSE;
		coil2 := FALSE;
		pre_heat := FALSE;
		ignite := FALSE;
		status := 5;
		last_change := tx;
	ELSIF NOT flame AND multiple_ignition THEN
		ignite := TRUE;
		state := 5;
		coil2 := FALSE;
		last_change := tx;
	ELSE
		IF tx - last_change >= post_ignite_time THEN
			(* post_ignite_time abgelaufen, ignite abschalten *)
			ignite := FALSE;
		END_IF;
		IF tx - last_change >= stage2_delay AND stage2 THEN
			coil2 := TRUE;
		ELSE
			coil2 := FALSE;
		END_IF;
	END_IF;
END_CASE;

(* abschaltung wenn kein eingangssignal *)
IF NOT in THEN
	state := 1;
	motor := FALSE;
	coil1 := FALSE;
	coil2 := FALSE;
	ignite := FALSE;
	pre_heat := FALSE;
	last_change := tx;
END_IF;

(* runtimezähler *)
timer1(in := flame AND in AND motor AND coil1 AND NOT coil2);
timer2(in := flame AND in AND motor AND coil1 AND coil2);
runtime1 := timer1.ontime;
runtime2 := timer2.ontime;
cycles := timer1.cycles;
KWH := runtime1 * KW1 + runtime2 * KW2;

(* zeit fuer naechsten aufruf merken *)
last := tx;

(* set fail output IF ERROR and Status  if normal operation *)

IF status > 0 AND status < 100 THEN
	fail := TRUE;
ELSE
	fail := FALSE;
	IF NOT in THEN
		status := 110;
	ELSIF flame AND in AND motor AND coil2 AND coil1 THEN
		status := 113;
	ELSIF flame AND in AND motor AND coil1 THEN
		status := 112;
	ELSE
		status := 111;
	END_IF;
END_IF;


(*
31.12.2006	hm		rev 1.1
	added pre_heat timing and output
	flame monitor before ignition will generate error on status output
	added output for KWh

31.12.2006	hm		rev 1.2
	added oil_temp_input

31.12.2006	hm		rev 1.3
	changed status output to be byte instead of bool

22.1.2007		hm		rev 1.4
	renamed fail output to status
	added output cycles
	corrected an error while pre_heat would be on when an error was present
	added coil2 output and stage2 input

15.9.2007		hm		rev 1.5
	replaced Time() with T_PLC_MS for compatibility and performance reasons

*)
END_FUNCTION_BLOCK

(* POU Byte_of_bit, ST *)
FUNCTION Byte_of_bit : BYTE
VAR_INPUT
	B0:BOOL;
	B1:BOOL;
	B2:BOOL;
	B3:BOOL;
	B4:BOOL;
	B5:BOOL;
	B6:BOOL;
	B7:BOOL;
END_VAR
VAR
	Bx : BYTE;
END_VAR

(*
version 1.0	4 aug 2006
programmer 	hugo
tested by		tobias

this function creates a byte from 8 individual bits

executioin TIME on wago 750-841 = 8 us
*)
BX.0 := B0;
BX.1 := B1;
BX.2 := B2;
BX.3 := B3;
BX.4 := B4;
BX.5 := B5;
BX.6 := B6;
BX.7 := B7;

Byte_of_bit := BX;
END_FUNCTION

(* POU Byte_of_Dword, ST *)
FUNCTION Byte_of_Dword : BYTE
VAR_INPUT
	in : DWORD;
	N : BYTE;
END_VAR
VAR
END_VAR

(*
version 1.1	2 jan 2008
programmer 	hugo
tested by		tobias

this function extracts a single byte from the nth position from right (right is lowest byte) 
the lower byte (starting with Bit0 from in) is selected with N=0.
*)
Byte_of_Dword := DWORD_TO_BYTE(SHR(in,n*8));

(* revision history
hm	17. jan 2007	rev 1.0
	original version

hm	2. jan 2008		rev 1.1
	improved performance

*)
END_FUNCTION

(* POU Byte_to_Bit, ST *)
FUNCTION_BLOCK Byte_to_Bit
VAR_INPUT
	IN: BYTE;
END_VAR
VAR_OUTPUT
	B0: BOOL;
	B1: BOOL;
	B2: BOOL;
	B3: BOOL;
	B4: BOOL;
	B5: BOOL;
	B6: BOOL;
	B7: BOOL;
END_VAR
VAR
END_VAR

(*
version 1.0	4 aug 2006
programmer 	hugo
tested by		tobias

this Function Block extracts the 8 Bits from a byte

executioin TIME on wago 750-841 = 13us
*)
B0 := IN.0;
B1 := IN.1;
B2 := IN.2;
B3 := IN.3;
B4 := IN.4;
B5 := IN.5;
B6 := IN.6;
B7 := IN.7;
END_FUNCTION_BLOCK

(* POU Byte_to_Range, ST *)
FUNCTION Byte_to_Range : REAL
VAR_INPUT
	X : BYTE;
	low : REAL;
	high : REAL;
END_VAR
VAR
END_VAR

(*
version 1.0	9. jan 2008
programmer 	hugo
tested by		tobias

Byte_to_Range converts a Byte into a real between low and high.

*)
Byte_to_Range := (high - low) * X / 255.0 + low;


(* revision history
hm	9. jan 2008		rev 1.0
	original version

*)
END_FUNCTION

(* POU BYTE_TO_STRB, ST *)
FUNCTION BYTE_TO_STRB : STRING
VAR_INPUT
	IN : BYTE;
END_VAR
VAR
	i: INT;
	pt : POINTER TO BYTE;
END_VAR

(*
version 1.1	15 dec 2007
programmer 	hugo
tested by		tobias

BYTE_TO_STRINGB converts a Byte to a String of Bits represented by '0' and '1' s.
The lowest order bit will be on the right and the high order bit on the left.

*)
(* pointer für die ausgabe ermitteln *)
pt := ADR(BYTE_TO_STRB);
(* die 8 ausgabecharacter ermitteln und schreiben *)
FOR i := 1 TO 8 DO
	IF in.7 THEN pt^ := 49; ELSE pt^ := 48; END_IF;
	in := SHL(in,1);
	pt := pt + 1;
END_FOR;

(* der ausgabestring muss noch mit 0 abgeschlossen werden *)
pt^ := 0;

(* code before rev 1.1
FOR i := 1 TO 8 DO
	IF in.0 = 0 THEN temp := CONCAT('0', temp); ELSE temp := CONCAT('1', temp); END_IF;
	in := SHR(in, 1);
END_FOR;
BYTE_TO_STRB := temp;
*)


(* revision history

hm		9.6.2007	rev 1.0		
	original version 

hm	15. dec 2007	rev 1.1
	inprooved code for higher performance

*)
END_FUNCTION

(* POU BYTE_TO_STRH, ST *)
FUNCTION BYTE_TO_STRH : STRING
VAR_INPUT
	IN : BYTE;
END_VAR
VAR
	temp : BYTE;
	PT : POINTER TO BYTE;
END_VAR

(*
version 1.2	15 dec 2007
programmer 	hugo
tested by		tobias

BYTE_TO_STRINGH converts a Byte to a String of Hexadecimal represented by '0' .. '9' and 'A' .. 'F'.
The lowest order Character will be on the right and the high order Character on the left.

*)
(* read pointer to output string *)
PT := ADR(BYTE_TO_STRH);
(* calculate high order hex value *)
temp := SHR(in,4);
(* convert value to hex character *)
IF temp <= 9 THEN temp := temp + 48; ELSE temp := temp + 55; END_IF;
(* write friat character to output string *)
PT^ := temp;
(* calculate low order hex value *)
temp := in AND 2#00001111;
IF temp <= 9 THEN temp := temp + 48; ELSE temp := temp + 55; END_IF;
(* increment pointer and wirte low order character *)
pt := pt + 1;
pt^ := temp;
(* set pointer at the end of the output string and close the string with 0 *)
pt := pt + 1;
pt^:= 0;


(* code before rev 1.2
FOR i := 1 TO 2 DO
	X := in AND 2#1111;
	IF X <= 9 THEN X := X + 48; ELSE X := X + 55; END_IF;
	Cx := CHR(X);
	temp := CONCAT(Cx, temp);
	in := SHR(in,4);
END_FOR;
BYTE_TO_STRH := temp;
*)

(* revision history

hm		9.6.2007		rev 1.0		
	original version 

hm		11.9.2007		rev 1.1		
	changed coding for compatibility with twincat, under twincat concat cannot have a function as argument.	

hm		15 dec 2007		REV 1.2
	changed code for higher performance
*)
END_FUNCTION

(* POU C_to_F, ST *)
FUNCTION C_to_F : REAL
VAR_INPUT
	celsius : REAL;
END_VAR
VAR
END_VAR

(*
version 1.0	4 aug 2006
programmer 	hugo
tested by		tobias

this function converts celsius  to fahrenheit 

*)
C_to_F := celsius * 1.8 + 32;
END_FUNCTION

(* POU C_to_K, ST *)
FUNCTION C_to_K : REAL
VAR_INPUT
	Celsius : REAL;
END_VAR
VAR
END_VAR

(*
version 1.0	4 dec 2006
programmer 	hugo
tested by		tobias

this function converts celsius to kelvin
*)
C_to_K := Celsius - 273.15;
END_FUNCTION

(* POU Calibrate, ST *)
FUNCTION_BLOCK Calibrate
VAR_INPUT
	X : REAL;
	CO : BOOL;
	CS : BOOL;
END_VAR
VAR_INPUT CONSTANT
	Y_Offset : REAL;
	Y_Scale : REAL;
END_VAR
VAR_OUTPUT
	Y : REAL;
END_VAR
VAR RETAIN
	offset : REAL;
	Scale : REAL := 1;
END_VAR

(*
	version 1.2	22 feb 2007
	programmer 	hugo
	tested BY		hans

Calibrate allows for offset and scale calibration of an analog input.
offset is calibrated to a stored reference Y_offset while CO is true.
after the offset is calibrated, scale can be calibrated to a reference value Y_scale while CS is true.
*)
(* check for calibration *)
IF CO THEN
	Offset := Y_Offset - X;
ELSIF CS THEN
	scale := Y_scale / (X+Offset);
END_IF;
(* calculate output *)
Y := (X + Offset) * Scale;


(* revision history
hm 22.2.2007		rev 1.2
	changed VAR RETAIN PERSISTENT to VAR RETAIN for better compatibility
	wago lon contollers do not support persisitent

*)
END_FUNCTION_BLOCK

(* POU ceil, ST *)
FUNCTION ceil : INT
VAR_INPUT
	X : REAL;
END_VAR
VAR
END_VAR


(*
version 1.0	7 feb 2007
programmer 	hugo
tested by		tobias

This is a rounding function which returns the smallest possible integer which is greater or equal to X.
ceil(3.14) = 4
ceil(-3.14) = -3

*)
ceil := TRUNC(X);
IF ceil < X THEN
	ceil := ceil + 1;
END_IF;
END_FUNCTION

(* POU check_parity, ST *)
FUNCTION check_parity : BOOL
VAR_INPUT
	in : DWORD;
	p : BOOL;
END_VAR
VAR
END_VAR

(*
version 1.2	8 dec 2007
programmer 	hugo
tested by		tobias

this function checks for an even partity for a dword and partity bit.

*)
check_parity := NOT p;
WHILE in > 0 DO
	check_parity := check_parity XOR in.0;
	in := SHR(in,1);
END_WHILE;

(* code before rev 1.2
WHILE in > 0 DO
	IF in.0 THEN cnt := cnt + 1; END_IF;
	in := SHR(in,1);
END_WHILE;
check_parity := even(cnt) XOR P;
*)


(* revision history

rev 1.0 HM  1.oct.2006

rev 1.1 hm	10.sep.2007
	changed algorithm to improove performance

rev 1.2	hm	8 dec 2007
	changed algorithm to improove performance
*)
END_FUNCTION

(* POU CHR, ST *)
FUNCTION CHR : STRING
VAR_INPUT
	C : BYTE;
END_VAR
VAR
	PT : POINTER TO BYTE;
END_VAR

(*
version 1.1	4. feb 2008
programmer 	hugo
tested by		tobias

CHR creates a character from a byte input and stuffs it in a one character length string.

*)
PT := ADR(CHR);
PT^ := C;
pt := pt + 1;
pt^ := 0;

(* revision history
hm		16 jan 2007		rev 1.0
	original version

hm		4. feb. 2008		rev 1.1
	return string would not be terminated properly
*)
END_FUNCTION

(* POU circle_A, ST *)
FUNCTION circle_A : REAL
VAR_INPUT
	rx : REAL;
	ax : REAL;
END_VAR
VAR
END_VAR

(*
version 1.1	4 dec 2007
programmer 	hugo
tested by		tobias

circle_A calculates the Area of a circle segement if ax = 360 the whole circle is calculated


*)
circle_A := PI1 * expn(Rx,2) / 360 * Ax;

(* revision histroy
hm	16. oct 2007	rev 1.0
	original version

hm	4. dec 2007		rev 1.1
	changed code for better performance
*)
END_FUNCTION

(* POU expn, ST *)
FUNCTION expn : REAL
VAR_INPUT
	X : REAL;
	N : INT;
END_VAR
VAR
END_VAR

(*
version 1.0	 2 dec 2007
programmer 	hugo
tested by		tobias

this function calculates X to the power of N (Y = X^N) whilke N is an integer
especially on CPU's without a floating point unit this algorythm is about 30 times faster then the IEC standard EXPT() Function

*)
IF n.15 THEN
	(* N is negative *)
	N := ABS(N);
	IF N.0 THEN expn := X; ELSE expn := 1; END_IF;
	N := SHR(N,1);
	WHILE N > 0 DO
		X := X * X;
		IF N.0 THEN expn := expn * X; END_IF;
		N := SHR(N,1);
	END_WHILE;
	expn := 1 / expn;
ELSE;
	IF N.0 THEN expn := X; ELSE expn := 1; END_IF;
	N := SHR(N,1);
	WHILE N > 0 DO
		X := X * X;
		IF N.0 THEN expn := expn * X; END_IF;
		N := SHR(N,1);
	END_WHILE;
END_IF;

(* revision history
hm	4. dec 2007		rev 1.0
	original version

*)
END_FUNCTION

(* POU circle_C, ST *)
FUNCTION circle_C : REAL
VAR_INPUT
	Rx : REAL;
	Ax : REAL;
END_VAR
VAR
END_VAR

(*
version 1.0	16 oct 2007
programmer 	hugo
tested by		tobias

circle_C calculates the Circumference of a circle  if ax = 360 the whole circle is calculated

*)
circle_C := PI2 * Rx * Ax / 360;

(* revision histroy
hm	16. oct 2007	rev 1.0
	original version

*)
END_FUNCTION

(* POU click, ST *)
FUNCTION_BLOCK click
VAR_INPUT
	in : BOOL;
END_VAR
VAR_OUTPUT
	Q : BOOL;
	single : BOOL;
	double : BOOL;
	triple : BOOL;
	status: BYTE;
END_VAR
VAR_INPUT CONSTANT
	T_debounce : TIME := t#10ms;
	T_short : TIME := t#200ms;
	T_pause : TIME := t#500ms;
	T_reconfig : TIME := t#1m;
END_VAR
VAR
	debounce : TON;
	tx : TIME;
	last : TIME;
	init : BOOL;
	edge : BOOL;
	standby: BOOL;
	state: INT;
END_VAR

(*
version 1.2	15 sep 2007
programmer 	oscat
tested by		tobias

click checks an input for single, double or tripple click and sets the corresponding output single, doulbe or triple for the time the input stays high at the last click.
the maximum high and low time for a click can beconfigrured with setup variables.
the input cinfigures itself to be high or low active dependung on which state the input stays longer than t_reconfig.

*)
(* read system time *)
tx := DWORD_TO_TIME(T_PLC_MS());

(* set last and tx if never started before *)
IF NOT init THEN
	init := TRUE;
	last := tx;
	debounce.PT := T_debounce;
	standby := in;
END_IF;

(* debounce input *)
debounce(in := in XOR standby);
Q := debounce.Q;

(* delete outputs if input is inactive *)
IF NOT Q THEN
	single := FALSE;
	double := FALSE;
	triple := FALSE;
	status := 110;
END_IF;

(* check for input edge *)
IF Q XOR edge THEN
	edge := in;
	last := tx;
	IF Q THEN state := state + 1; END_IF;
END_IF;

IF (q AND tx - last >= T_short) OR (NOT q AND tx - last >= t_pause) THEN
	CASE state OF
		1:	single := TRUE;
			status := 111;
		2:	double := TRUE;
			status := 112;
		3:	triple := TRUE;
			status := 113;
	END_CASE;
	state := 0;
END_IF;

(* determine if high or low active *)
IF tx - last >= t_reconfig THEN
	standby := in;
	last := tx;
END_IF;



(* revision history

15 Feb 2007	rev 1.0	hm
	created original version

18.5.2007		rev 1.1 hm
	corrected an error while execution would stop after t_reconfig elapsed.

15.9.2007		rev 1.2 hm
	replaced Time() with T_PLC_MS for compatibility and performance reasons

*)
END_FUNCTION_BLOCK

(* POU clk_div, ST *)
FUNCTION_BLOCK clk_div
VAR_INPUT
	clk : BOOL;
	rst: BOOL;
END_VAR
VAR_OUTPUT
	Q0 : BOOL := 0;
	Q1 : BOOL := 0;
	Q2 : BOOL := 0;
	Q3 : BOOL := 0;
	Q4 : BOOL := 0;
	Q5 : BOOL := 0;
	Q6 : BOOL := 0;
	Q7 : BOOL := 0;
END_VAR
VAR
	cnt: BYTE := 0;
END_VAR

(*
version 1.1	2 jan 2008
programmer 	hugo
tested by		tobias

this is a clock divider
each output divides the signal by 2
Q0 = clk / 2 , Q1 = Q0 / 2 and so on.
the outputs have a 50% duty cycle each.


*)
IF rst THEN
	cnt:= 0;
	Q0 := 0;
	Q1 := 0;
	Q2 := 0;
	Q3 := 0;
	Q4 := 0;
	Q5 := 0;
	Q6 := 0;
	Q7 := 0;
ELSIF clk THEN
	cnt:= cnt +1;
	Q0 := cnt.0;
	Q1 := cnt.1;
	Q2 := cnt.2;
	Q3 := cnt.3;
	Q4 := cnt.4;
	Q5 := cnt.5;
	Q6 := cnt.6;
	Q7 := cnt.7;
END_IF;

(* revision history
hm	4. aug. 2006	rev 1.0
	original version

hm	2. jan 2008		rev 1.1
	improved performance

*)
END_FUNCTION_BLOCK

(* POU CLK_N, ST *)
FUNCTION_BLOCK CLK_N
VAR_INPUT
	N : INT;
END_VAR
VAR_OUTPUT
	Q : BOOL;
END_VAR
VAR
	edge : BOOL := 0;
	stime: DWORD;
	clk: BOOL;
END_VAR

(*
version 1.0	17 sep 2007
programmer 	hugo
tested by		tobias

clk_N uses the internal sps time to generate one pulse every N ms
every pulse is only valid for one cycle so that a edge trigger is not necessary
clk_N generates pulses depending on the accuracy of the system clock.
The input N controlls the period time of the clock.
N=0 equals 1ms, N=1 equals 2ms, N=2 equals 4ms, N=3 equals 8ms ....

be careful, 1ms clocks will only work on very powerful sps cpu's
*)
stime := SHR(T_PLC_MS(),N);
clk := stime.0;
Q := clk XOR edge;
edge := CLK;

(* revision history
hm	16. dec 2007		rev 1.0
	original version

*)
END_FUNCTION_BLOCK

(* POU CLK_Prg, ST *)
	FUNCTION_BLOCK CLK_Prg
VAR_INPUT
	PT : TIME := t#10ms;
END_VAR
VAR_OUTPUT
	Q : BOOL := 0;
END_VAR
VAR
	init : BOOL := FALSE;
	last : TIME;
	tx: TIME;
END_VAR

(*
version 1.2	17 sep 2007
programmer 	hugo
tested by		tobias

clk_prg uses the internal sps time to generate a clock with programmable period time.
the period time is defined for 10ms .. 65s
the first cycle after start is a clk pulse and then depending on the programmed period time a delay.
every pulse is only valid for one cycle.
the accuracy of clk_prg is depending on the accuracy of the system clock.

*)
(* read system time *)
tx := DWORD_TO_TIME(T_PLC_MS());

(* initialize on startup *)
IF NOT init THEN
	init := TRUE;
	last := tx - pt;
END_IF;

(* generate output pulse when next_pulse is reached *)
IF tx - last >= pt THEN
	Q := TRUE;
	last := tx;
ELSE
	Q := FALSE;
END_IF;


(* revision hiostory

hm 25 feb 2007	rev 1.1
	rewritten code for higher performance
	pt can now be changed during runtime

hm	17. sep 2007	rev 1.2
	replaced time() with t_plc_ms() for compatibility reasons

*)
END_FUNCTION_BLOCK

(* POU CLK_Pulse, ST *)
FUNCTION_BLOCK CLK_Pulse
VAR_INPUT
	PT : TIME := t#10ms;
	N : INT := 0;
	rst : BOOL := 0;
END_VAR
VAR_OUTPUT
	Q : BOOL := 0;
	cnt : INT := 0;
	run : BOOL := 0;
END_VAR
VAR
	pti : TIME := t#0ms;
	next_pulse: TIME := T#0s;
	overflow: BOOL := FALSE;
	tx: TIME;
END_VAR

(*
version 1.1	17 sep 2007
programmer 	hugo
tested by		tobias

clk_pulse uses the internal sps time to generate a clock with programmable period time.
the period time is defined for 10ms .. 65s.
pulse generation is continuous if N = 0 and for n pulses otherwise.
if the period time is set to less then 10ms the min clock perid is 10ms.
the first cycle after start is a clk pulse and then depending on the programmed period time a delay.
every pulse is only valid for one cycle so that a edge trigger is not necessary
clk_prg depending on the accuracy of the system clock.

*)
(* read system *)
tx := DWORD_TO_TIME(T_PLC_MS());


IF rst THEN
	run := FALSE;
	pti := t#0ms;
	next_pulse := t#0ms;
	overflow := FALSE;
	Q := FALSE;
	cnt := 0;
ELSIF cnt <= N OR N = 0 THEN
	IF NOT run THEN
		next_pulse := tx;
		run := TRUE;
		IF pt < T#10ms THEN PTI := T#10ms; ELSE pti := pt; END_IF;
	END_IF;
	IF tx >= next_pulse AND NOT overflow AND (cnt < N OR N = 0) THEN
		Q := TRUE;
		cnt := cnt + 1;
		IF next_pulse + pti < next_pulse THEN
			overflow := TRUE;
		END_IF;
		next_pulse := next_pulse + pti;
	ELSE
		Q := FALSE;
		IF cnt = N THEN run := FALSE; END_IF
		IF tx <= next_pulse THEN overflow := FALSE; END_IF;
	END_IF;
END_IF

(* revision history
hm		4. aug 2006		rev 1.0
	original version

hm		17. sep 2007	rev 1.1
	replaced time() with T_PLC_S() fr compatblity reasons

*)
END_FUNCTION_BLOCK

(* POU cone_V, ST *)
FUNCTION cone_V : REAL
VAR_INPUT
	rx : REAL;
	hx : REAL;
END_VAR
VAR
END_VAR

(*
version 1.1	4 dec 2007
programmer 	hugo
tested by		tobias

cone_V calculates the Volume of a cone

*)
cone_V := PI1 / 3 * expn(Rx,2) * hx;

